DATA_BLOCK "DB_Result"
{ S7_Optimized_Access := 'TRUE' }
VERSION : 0.1
NON_RETAIN
   VAR
      TruePositive : Int;
      TrueNegative : Int;
      FalsePositive : Int;
      FalseNegative : Int;
      Predicted_class : Int;
      MismatchCount : Int;
      EXPECTED_TRUE_NEGATIVE : Int;
      EXPECTED_FALSE_POSITIVE : Int;
      EXPECTED_FALSE_NEGATIVE : Int;
      EXPECTED_TRUE_POSITIVE : Int;
      EXPECTED_PREDICITON_COUNT : Int;
      THRESHOLD : Real;
   END_VAR


BEGIN
   EXPECTED_TRUE_NEGATIVE := 1648;
   EXPECTED_FALSE_POSITIVE := 106;
   EXPECTED_FALSE_NEGATIVE := 55;
   EXPECTED_TRUE_POSITIVE := 885;
   EXPECTED_PREDICITON_COUNT := 2694;
   THRESHOLD := 0.05268643;

END_DATA_BLOCK

DATA_BLOCK "DB_Main"
{ S7_Optimized_Access := 'TRUE' }
VERSION : 0.1
NON_RETAIN
   VAR
      iState : Int;
      PredictCount : Int;
      bStart : Bool;
      Mse : Real;
   END_VAR


BEGIN

END_DATA_BLOCK

DATA_BLOCK "DB_Attack_v0_first_attack"
{ S7_Optimized_Access := 'TRUE' }
VERSION : 0.1
NON_RETAIN
   VAR
      DATA : Array[0..2693, 0..40] of Real;
   END_VAR


BEGIN
   DATA[0,0] := 2.427057;
   DATA[0,1] := 522.8467;
   DATA[0,2] := 2.0;
   DATA[0,3] := 2.0;
   DATA[0,4] := 262.0161;
   DATA[0,5] := 8.396437;
   DATA[0,6] := 328.6337;
   DATA[0,7] := 2.445391;
   DATA[0,8] := 2.0;
   DATA[0,9] := 2.0;
   DATA[0,10] := 2.0;
   DATA[0,11] := 19.74838;
   DATA[0,12] := 2.206835;
   DATA[0,13] := 956.1651;
   DATA[0,14] := 1.0;
   DATA[0,15] := 2.0;
   DATA[0,16] := 1.0;
   DATA[0,17] := 1.0;
   DATA[0,18] := 1.0;
   DATA[0,19] := 2.0;
   DATA[0,20] := 148.808;
   DATA[0,21] := 156.0882;
   DATA[0,22] := 1.713517;
   DATA[0,23] := 942.0662;
   DATA[0,24] := 2.0;
   DATA[0,25] := 2.0;
   DATA[0,26] := 7.878621;
   DATA[0,27] := 145.1166;
   DATA[0,28] := 264.5475;
   DATA[0,29] := 12.03538;
   DATA[0,30] := 1.723789;
   DATA[0,31] := 1.279621;
   DATA[0,32] := 0.7352687;
   DATA[0,33] := 0.3077859;
   DATA[0,34] := 2.0;
   DATA[0,35] := 250.8652;
   DATA[0,36] := 1.649953;
   DATA[0,37] := 189.5988;
   DATA[0,38] := 0.000128152;
   DATA[0,39] := 1.0;
   DATA[1,0] := 2.446274;
   DATA[1,1] := 522.886;
   DATA[1,2] := 2.0;
   DATA[1,3] := 2.0;
   DATA[1,4] := 262.0161;
   DATA[1,5] := 8.396437;
   DATA[1,6] := 328.6337;
   DATA[1,7] := 2.445391;
   DATA[1,8] := 2.0;
   DATA[1,9] := 2.0;
   DATA[1,10] := 2.0;
   DATA[1,11] := 19.74838;
   DATA[1,12] := 2.208244;
   DATA[1,13] := 956.1651;
   DATA[1,14] := 1.0;
   DATA[1,15] := 2.0;
   DATA[1,16] := 1.0;
   DATA[1,17] := 1.0;
   DATA[1,18] := 1.0;
   DATA[1,19] := 2.0;
   DATA[1,20] := 148.808;
   DATA[1,21] := 156.0882;
   DATA[1,22] := 1.715952;
   DATA[1,23] := 942.0277;
   DATA[1,24] := 2.0;
   DATA[1,25] := 2.0;
   DATA[1,26] := 7.878621;
   DATA[1,27] := 145.1166;
   DATA[1,28] := 264.5475;
   DATA[1,29] := 12.03538;
   DATA[1,30] := 1.723789;
   DATA[1,31] := 1.297554;
   DATA[1,32] := 0.7352687;
   DATA[1,33] := 0.3077859;
   DATA[1,34] := 2.0;
   DATA[1,35] := 250.8652;
   DATA[1,36] := 1.649953;
   DATA[1,37] := 189.6789;
   DATA[1,38] := 0.000128152;
   DATA[1,39] := 1.0;
   DATA[2,0] := 2.489191;
   DATA[2,1] := 522.8467;
   DATA[2,2] := 2.0;
   DATA[2,3] := 2.0;
   DATA[2,4] := 262.0161;
   DATA[2,5] := 8.394514;
   DATA[2,6] := 328.6337;
   DATA[2,7] := 2.442316;
   DATA[2,8] := 2.0;
   DATA[2,9] := 2.0;
   DATA[2,10] := 2.0;
   DATA[2,11] := 19.69076;
   DATA[2,12] := 2.208628;
   DATA[2,13] := 956.4855;
   DATA[2,14] := 1.0;
   DATA[2,15] := 2.0;
   DATA[2,16] := 1.0;
   DATA[2,17] := 1.0;
   DATA[2,18] := 1.0;
   DATA[2,19] := 2.0;
   DATA[2,20] := 148.808;
   DATA[2,21] := 156.0882;
   DATA[2,22] := 1.715952;
   DATA[2,23] := 941.8739;
   DATA[2,24] := 2.0;
   DATA[2,25] := 2.0;
   DATA[2,26] := 7.878621;
   DATA[2,27] := 145.1166;
   DATA[2,28] := 264.5475;
   DATA[2,29] := 12.03538;
   DATA[2,30] := 1.723404;
   DATA[2,31] := 1.293967;
   DATA[2,32] := 0.7352687;
   DATA[2,33] := 0.3086186;
   DATA[2,34] := 2.0;
   DATA[2,35] := 250.8812;
   DATA[2,36] := 1.649953;
   DATA[2,37] := 189.6789;
   DATA[2,38] := 0.000128152;
   DATA[2,39] := 1.0;
   DATA[3,0] := 2.53435;
   DATA[3,1] := 522.9645;
   DATA[3,2] := 2.0;
   DATA[3,3] := 2.0;
   DATA[3,4] := 262.0161;
   DATA[3,5] := 8.394514;
   DATA[3,6] := 328.6337;
   DATA[3,7] := 2.442316;
   DATA[3,8] := 2.0;
   DATA[3,9] := 2.0;
   DATA[3,10] := 2.0;
   DATA[3,11] := 19.69076;
   DATA[3,12] := 2.208628;
   DATA[3,13] := 956.806;
   DATA[3,14] := 1.0;
   DATA[3,15] := 2.0;
   DATA[3,16] := 1.0;
   DATA[3,17] := 1.0;
   DATA[3,18] := 1.0;
   DATA[3,19] := 2.0;
   DATA[3,20] := 148.808;
   DATA[3,21] := 156.0882;
   DATA[3,22] := 1.71467;
   DATA[3,23] := 941.797;
   DATA[3,24] := 2.0;
   DATA[3,25] := 2.0;
   DATA[3,26] := 7.878621;
   DATA[3,27] := 145.0141;
   DATA[3,28] := 264.5475;
   DATA[3,29] := 12.03538;
   DATA[3,30] := 1.723404;
   DATA[3,31] := 1.281158;
   DATA[3,32] := 0.7352687;
   DATA[3,33] := 0.3086186;
   DATA[3,34] := 2.0;
   DATA[3,35] := 250.8812;
   DATA[3,36] := 1.649953;
   DATA[3,37] := 189.6148;
   DATA[3,38] := 0.000128152;
   DATA[3,39] := 1.0;
   DATA[4,0] := 2.56926;
   DATA[4,1] := 523.4748;
   DATA[4,2] := 2.0;
   DATA[4,3] := 2.0;
   DATA[4,4] := 262.0161;
   DATA[4,5] := 8.394514;
   DATA[4,6] := 328.6337;
   DATA[4,7] := 2.443085;
   DATA[4,8] := 2.0;
   DATA[4,9] := 2.0;
   DATA[4,10] := 2.0;
   DATA[4,11] := 19.69076;
   DATA[4,12] := 2.208628;
   DATA[4,13] := 957.0864;
   DATA[4,14] := 1.0;
   DATA[4,15] := 2.0;
   DATA[4,16] := 1.0;
   DATA[4,17] := 1.0;
   DATA[4,18] := 1.0;
   DATA[4,19] := 2.0;
   DATA[4,20] := 148.808;
   DATA[4,21] := 156.0882;
   DATA[4,22] := 1.71467;
   DATA[4,23] := 942.22;
   DATA[4,24] := 2.0;
   DATA[4,25] := 2.0;
   DATA[4,26] := 7.878621;
   DATA[4,27] := 144.8859;
   DATA[4,28] := 264.5475;
   DATA[4,29] := 12.03538;
   DATA[4,30] := 1.723404;
   DATA[4,31] := 1.281158;
   DATA[4,32] := 0.7352687;
   DATA[4,33] := 0.3086186;
   DATA[4,34] := 2.0;
   DATA[4,35] := 250.8812;
   DATA[4,36] := 1.649953;
   DATA[4,37] := 189.5027;
   DATA[4,38] := 0.000128152;
   DATA[4,39] := 1.0;
   DATA[5,0] := 2.609294;
   DATA[5,1] := 523.8673;
   DATA[5,2] := 2.0;
   DATA[5,3] := 2.0;
   DATA[5,4] := 262.0161;
   DATA[5,5] := 8.394514;
   DATA[5,6] := 328.6337;
   DATA[5,7] := 2.44411;
   DATA[5,8] := 2.0;
   DATA[5,9] := 2.0;
   DATA[5,10] := 2.0;
   DATA[5,11] := 19.69076;
   DATA[5,12] := 2.207347;
   DATA[5,13] := 957.1664;
   DATA[5,14] := 1.0;
   DATA[5,15] := 2.0;
   DATA[5,16] := 1.0;
   DATA[5,17] := 1.0;
   DATA[5,18] := 1.0;
   DATA[5,19] := 2.0;
   DATA[5,20] := 148.808;
   DATA[5,21] := 155.96;
   DATA[5,22] := 1.71467;
   DATA[5,23] := 942.6429;
   DATA[5,24] := 2.0;
   DATA[5,25] := 2.0;
   DATA[5,26] := 7.878621;
   DATA[5,27] := 144.8859;
   DATA[5,28] := 264.5475;
   DATA[5,29] := 12.03538;
   DATA[5,30] := 1.723404;
   DATA[5,31] := 1.272704;
   DATA[5,32] := 0.7352687;
   DATA[5,33] := 0.3086186;
   DATA[5,34] := 2.0;
   DATA[5,35] := 250.753;
   DATA[5,36] := 1.649953;
   DATA[5,37] := 189.5027;
   DATA[5,38] := 0.000128152;
   DATA[5,39] := 1.0;
   DATA[6,0] := 2.637158;
   DATA[6,1] := 524.1028;
   DATA[6,2] := 2.0;
   DATA[6,3] := 2.0;
   DATA[6,4] := 262.0161;
   DATA[6,5] := 8.394514;
   DATA[6,6] := 328.6337;
   DATA[6,7] := 2.44411;
   DATA[6,8] := 2.0;
   DATA[6,9] := 2.0;
   DATA[6,10] := 2.0;
   DATA[6,11] := 19.69076;
   DATA[6,12] := 2.210037;
   DATA[6,13] := 957.0062;
   DATA[6,14] := 1.0;
   DATA[6,15] := 2.0;
   DATA[6,16] := 1.0;
   DATA[6,17] := 1.0;
   DATA[6,18] := 1.0;
   DATA[6,19] := 2.0;
   DATA[6,20] := 148.808;
   DATA[6,21] := 155.96;
   DATA[6,22] := 1.713004;
   DATA[6,23] := 942.7582;
   DATA[6,24] := 2.0;
   DATA[6,25] := 2.0;
   DATA[6,26] := 7.878621;
   DATA[6,27] := 144.8859;
   DATA[6,28] := 264.5475;
   DATA[6,29] := 12.03538;
   DATA[6,30] := 1.723404;
   DATA[6,31] := 1.270142;
   DATA[6,32] := 0.7352687;
   DATA[6,33] := 0.3086186;
   DATA[6,34] := 2.0;
   DATA[6,35] := 250.5928;
   DATA[6,36] := 1.649953;
   DATA[6,37] := 189.5027;
   DATA[6,38] := 0.000128152;
   DATA[6,39] := 1.0;
   DATA[7,0] := 2.652211;
   DATA[7,1] := 524.2206;
   DATA[7,2] := 2.0;
   DATA[7,3] := 2.0;
   DATA[7,4] := 262.0161;
   DATA[7,5] := 8.394514;
   DATA[7,6] := 328.6337;
   DATA[7,7] := 2.441803;
   DATA[7,8] := 2.0;
   DATA[7,9] := 2.0;
   DATA[7,10] := 2.0;
   DATA[7,11] := 19.69076;
   DATA[7,12] := 2.210037;
   DATA[7,13] := 957.2866;
   DATA[7,14] := 1.0;
   DATA[7,15] := 2.0;
   DATA[7,16] := 1.0;
   DATA[7,17] := 1.0;
   DATA[7,18] := 1.0;
   DATA[7,19] := 2.0;
   DATA[7,20] := 148.808;
   DATA[7,21] := 155.96;
   DATA[7,22] := 1.713004;
   DATA[7,23] := 943.1043;
   DATA[7,24] := 2.0;
   DATA[7,25] := 2.0;
   DATA[7,26] := 7.878621;
   DATA[7,27] := 144.8859;
   DATA[7,28] := 264.5475;
   DATA[7,29] := 12.03538;
   DATA[7,30] := 1.723404;
   DATA[7,31] := 1.262329;
   DATA[7,32] := 0.7352687;
   DATA[7,33] := 0.3086186;
   DATA[7,34] := 2.0;
   DATA[7,35] := 250.5928;
   DATA[7,36] := 1.649953;
   DATA[7,37] := 189.5027;
   DATA[7,38] := 0.000128152;
   DATA[7,39] := 1.0;
   DATA[8,0] := 2.655735;
   DATA[8,1] := 524.4954;
   DATA[8,2] := 2.0;
   DATA[8,3] := 2.0;
   DATA[8,4] := 262.0161;
   DATA[8,5] := 8.394514;
   DATA[8,6] := 328.6337;
   DATA[8,7] := 2.441803;
   DATA[8,8] := 2.0;
   DATA[8,9] := 2.0;
   DATA[8,10] := 2.0;
   DATA[8,11] := 19.66195;
   DATA[8,12] := 2.210037;
   DATA[8,13] := 957.6071;
   DATA[8,14] := 1.0;
   DATA[8,15] := 2.0;
   DATA[8,16] := 1.0;
   DATA[8,17] := 1.0;
   DATA[8,18] := 1.0;
   DATA[8,19] := 2.0;
   DATA[8,20] := 148.808;
   DATA[8,21] := 155.96;
   DATA[8,22] := 1.71262;
   DATA[8,23] := 943.3735;
   DATA[8,24] := 2.0;
   DATA[8,25] := 2.0;
   DATA[8,26] := 7.878621;
   DATA[8,27] := 144.8859;
   DATA[8,28] := 264.5475;
   DATA[8,29] := 12.03538;
   DATA[8,30] := 1.723404;
   DATA[8,31] := 1.270398;
   DATA[8,32] := 0.7352687;
   DATA[8,33] := 0.3086186;
   DATA[8,34] := 2.0;
   DATA[8,35] := 250.9132;
   DATA[8,36] := 1.649953;
   DATA[8,37] := 189.5027;
   DATA[8,38] := 0.000128152;
   DATA[8,39] := 1.0;
   DATA[9,0] := 2.64997;
   DATA[9,1] := 524.0636;
   DATA[9,2] := 2.0;
   DATA[9,3] := 2.0;
   DATA[9,4] := 262.0161;
   DATA[9,5] := 8.394514;
   DATA[9,6] := 328.6337;
   DATA[9,7] := 2.441803;
   DATA[9,8] := 2.0;
   DATA[9,9] := 2.0;
   DATA[9,10] := 2.0;
   DATA[9,11] := 19.66195;
   DATA[9,12] := 2.210037;
   DATA[9,13] := 957.2866;
   DATA[9,14] := 1.0;
   DATA[9,15] := 2.0;
   DATA[9,16] := 1.0;
   DATA[9,17] := 1.0;
   DATA[9,18] := 1.0;
   DATA[9,19] := 2.0;
   DATA[9,20] := 148.808;
   DATA[9,21] := 155.96;
   DATA[9,22] := 1.71262;
   DATA[9,23] := 943.6042;
   DATA[9,24] := 2.0;
   DATA[9,25] := 2.0;
   DATA[9,26] := 7.878621;
   DATA[9,27] := 144.8859;
   DATA[9,28] := 264.5475;
   DATA[9,29] := 12.03538;
   DATA[9,30] := 1.726224;
   DATA[9,31] := 1.281158;
   DATA[9,32] := 0.7352687;
   DATA[9,33] := 0.3084905;
   DATA[9,34] := 2.0;
   DATA[9,35] := 250.9132;
   DATA[9,36] := 1.649953;
   DATA[9,37] := 189.5668;
   DATA[9,38] := 0.000128152;
   DATA[9,39] := 1.0;
   DATA[10,0] := 2.630433;
   DATA[10,1] := 524.1028;
   DATA[10,2] := 2.0;
   DATA[10,3] := 2.0;
   DATA[10,4] := 262.0161;
   DATA[10,5] := 8.394514;
   DATA[10,6] := 328.6337;
   DATA[10,7] := 2.441803;
   DATA[10,8] := 2.0;
   DATA[10,9] := 2.0;
   DATA[10,10] := 2.0;
   DATA[10,11] := 19.68756;
   DATA[10,12] := 2.210037;
   DATA[10,13] := 957.6071;
   DATA[10,14] := 1.0;
   DATA[10,15] := 2.0;
   DATA[10,16] := 1.0;
   DATA[10,17] := 1.0;
   DATA[10,18] := 1.0;
   DATA[10,19] := 2.0;
   DATA[10,20] := 148.808;
   DATA[10,21] := 155.96;
   DATA[10,22] := 1.715439;
   DATA[10,23] := 943.9118;
   DATA[10,24] := 2.0;
   DATA[10,25] := 2.0;
   DATA[10,26] := 7.878621;
   DATA[10,27] := 144.8859;
   DATA[10,28] := 264.5475;
   DATA[10,29] := 12.03538;
   DATA[10,30] := 1.726352;
   DATA[10,31] := 1.276162;
   DATA[10,32] := 0.7352687;
   DATA[10,33] := 0.3081062;
   DATA[10,34] := 2.0;
   DATA[10,35] := 251.1055;
   DATA[10,36] := 1.649953;
   DATA[10,37] := 189.8231;
   DATA[10,38] := 0.000128152;
   DATA[10,39] := 1.0;
   DATA[11,0] := 2.621785;
   DATA[11,1] := 523.7496;
   DATA[11,2] := 2.0;
   DATA[11,3] := 2.0;
   DATA[11,4] := 262.0161;
   DATA[11,5] := 8.391951;
   DATA[11,6] := 328.6337;
   DATA[11,7] := 2.441803;
   DATA[11,8] := 2.0;
   DATA[11,9] := 2.0;
   DATA[11,10] := 2.0;
   DATA[11,11] := 19.72598;
   DATA[11,12] := 2.210037;
   DATA[11,13] := 957.2065;
   DATA[11,14] := 1.0;
   DATA[11,15] := 2.0;
   DATA[11,16] := 1.0;
   DATA[11,17] := 1.0;
   DATA[11,18] := 1.0;
   DATA[11,19] := 2.0;
   DATA[11,20] := 148.808;
   DATA[11,21] := 156.1138;
   DATA[11,22] := 1.716721;
   DATA[11,23] := 943.9118;
   DATA[11,24] := 2.0;
   DATA[11,25] := 2.0;
   DATA[11,26] := 7.878621;
   DATA[11,27] := 144.8859;
   DATA[11,28] := 264.5475;
   DATA[11,29] := 12.03538;
   DATA[11,30] := 1.726352;
   DATA[11,31] := 1.282183;
   DATA[11,32] := 0.7352687;
   DATA[11,33] := 0.3074016;
   DATA[11,34] := 2.0;
   DATA[11,35] := 251.1856;
   DATA[11,36] := 1.649953;
   DATA[11,37] := 189.9994;
   DATA[11,38] := 0.000128152;
   DATA[11,39] := 1.0;
   DATA[12,0] := 2.61602;
   DATA[12,1] := 523.4355;
   DATA[12,2] := 2.0;
   DATA[12,3] := 2.0;
   DATA[12,4] := 262.0161;
   DATA[12,5] := 8.390669;
   DATA[12,6] := 328.6337;
   DATA[12,7] := 2.441803;
   DATA[12,8] := 2.0;
   DATA[12,9] := 2.0;
   DATA[12,10] := 2.0;
   DATA[12,11] := 19.75479;
   DATA[12,12] := 2.210037;
   DATA[12,13] := 957.5269;
   DATA[12,14] := 1.0;
   DATA[12,15] := 2.0;
   DATA[12,16] := 1.0;
   DATA[12,17] := 1.0;
   DATA[12,18] := 1.0;
   DATA[12,19] := 2.0;
   DATA[12,20] := 148.808;
   DATA[12,21] := 156.1138;
   DATA[12,22] := 1.717874;
   DATA[12,23] := 944.181;
   DATA[12,24] := 2.0;
   DATA[12,25] := 2.0;
   DATA[12,26] := 7.878621;
   DATA[12,27] := 144.8859;
   DATA[12,28] := 264.5475;
   DATA[12,29] := 12.03538;
   DATA[12,30] := 1.72725;
   DATA[12,31] := 1.275778;
   DATA[12,32] := 0.7352687;
   DATA[12,33] := 0.3066329;
   DATA[12,34] := 2.0;
   DATA[12,35] := 251.1856;
   DATA[12,36] := 1.649953;
   DATA[12,37] := 189.9994;
   DATA[12,38] := 0.000128152;
   DATA[12,39] := 1.0;
   DATA[13,0] := 2.599366;
   DATA[13,1] := 523.043;
   DATA[13,2] := 2.0;
   DATA[13,3] := 2.0;
   DATA[13,4] := 262.0161;
   DATA[13,5] := 8.390669;
   DATA[13,6] := 328.6337;
   DATA[13,7] := 2.441803;
   DATA[13,8] := 2.0;
   DATA[13,9] := 2.0;
   DATA[13,10] := 2.0;
   DATA[13,11] := 19.79;
   DATA[13,12] := 2.210037;
   DATA[13,13] := 957.8875;
   DATA[13,14] := 1.0;
   DATA[13,15] := 2.0;
   DATA[13,16] := 1.0;
   DATA[13,17] := 1.0;
   DATA[13,18] := 1.0;
   DATA[13,19] := 2.0;
   DATA[13,20] := 148.808;
   DATA[13,21] := 156.1138;
   DATA[13,22] := 1.717874;
   DATA[13,23] := 943.9118;
   DATA[13,24] := 2.0;
   DATA[13,25] := 2.0;
   DATA[13,26] := 7.878621;
   DATA[13,27] := 144.8859;
   DATA[13,28] := 264.5475;
   DATA[13,29] := 12.03538;
   DATA[13,30] := 1.728275;
   DATA[13,31] := 1.272192;
   DATA[13,32] := 0.7352687;
   DATA[13,33] := 0.3066329;
   DATA[13,34] := 2.0;
   DATA[13,35] := 251.1856;
   DATA[13,36] := 1.649953;
   DATA[13,37] := 189.9994;
   DATA[13,38] := 0.000128152;
   DATA[13,39] := 1.0;
   DATA[14,0] := 2.588476;
   DATA[14,1] := 522.729;
   DATA[14,2] := 2.0;
   DATA[14,3] := 2.0;
   DATA[14,4] := 262.0161;
   DATA[14,5] := 8.390669;
   DATA[14,6] := 328.6337;
   DATA[14,7] := 2.441803;
   DATA[14,8] := 2.0;
   DATA[14,9] := 2.0;
   DATA[14,10] := 2.0;
   DATA[14,11] := 19.79;
   DATA[14,12] := 2.209525;
   DATA[14,13] := 958.288;
   DATA[14,14] := 1.0;
   DATA[14,15] := 2.0;
   DATA[14,16] := 1.0;
   DATA[14,17] := 1.0;
   DATA[14,18] := 1.0;
   DATA[14,19] := 2.0;
   DATA[14,20] := 148.808;
   DATA[14,21] := 156.1138;
   DATA[14,22] := 1.717874;
   DATA[14,23] := 943.9887;
   DATA[14,24] := 2.0;
   DATA[14,25] := 2.0;
   DATA[14,26] := 7.878621;
   DATA[14,27] := 144.8859;
   DATA[14,28] := 264.5475;
   DATA[14,29] := 12.26609;
   DATA[14,30] := 1.728275;
   DATA[14,31] := 1.282951;
   DATA[14,32] := 0.7352687;
   DATA[14,33] := 0.3066329;
   DATA[14,34] := 2.0;
   DATA[14,35] := 251.1856;
   DATA[14,36] := 1.649953;
   DATA[14,37] := 189.9994;
   DATA[14,38] := 0.000128152;
   DATA[14,39] := 1.0;
   DATA[15,0] := 2.567979;
   DATA[15,1] := 522.6505;
   DATA[15,2] := 2.0;
   DATA[15,3] := 2.0;
   DATA[15,4] := 262.0161;
   DATA[15,5] := 8.390669;
   DATA[15,6] := 328.6337;
   DATA[15,7] := 2.441803;
   DATA[15,8] := 2.0;
   DATA[15,9] := 2.0;
   DATA[15,10] := 2.0;
   DATA[15,11] := 19.73878;
   DATA[15,12] := 2.209525;
   DATA[15,13] := 958.288;
   DATA[15,14] := 1.0;
   DATA[15,15] := 2.0;
   DATA[15,16] := 1.0;
   DATA[15,17] := 1.0;
   DATA[15,18] := 1.0;
   DATA[15,19] := 2.0;
   DATA[15,20] := 148.808;
   DATA[15,21] := 156.1138;
   DATA[15,22] := 1.717874;
   DATA[15,23] := 944.4117;
   DATA[15,24] := 2.0;
   DATA[15,25] := 2.0;
   DATA[15,26] := 7.878621;
   DATA[15,27] := 144.8859;
   DATA[15,28] := 264.5475;
   DATA[15,29] := 12.26609;
   DATA[15,30] := 1.728275;
   DATA[15,31] := 1.282951;
   DATA[15,32] := 0.7352687;
   DATA[15,33] := 0.3066329;
   DATA[15,34] := 2.0;
   DATA[15,35] := 251.1856;
   DATA[15,36] := 1.649953;
   DATA[15,37] := 189.9994;
   DATA[15,38] := 0.000128152;
   DATA[15,39] := 1.0;
   DATA[16,0] := 2.556769;
   DATA[16,1] := 522.6897;
   DATA[16,2] := 2.0;
   DATA[16,3] := 2.0;
   DATA[16,4] := 262.0161;
   DATA[16,5] := 8.390669;
   DATA[16,6] := 328.6337;
   DATA[16,7] := 2.441803;
   DATA[16,8] := 2.0;
   DATA[16,9] := 2.0;
   DATA[16,10] := 2.0;
   DATA[16,11] := 19.70997;
   DATA[16,12] := 2.207091;
   DATA[16,13] := 958.5684;
   DATA[16,14] := 1.0;
   DATA[16,15] := 2.0;
   DATA[16,16] := 1.0;
   DATA[16,17] := 1.0;
   DATA[16,18] := 1.0;
   DATA[16,19] := 2.0;
   DATA[16,20] := 148.808;
   DATA[16,21] := 156.1138;
   DATA[16,22] := 1.717874;
   DATA[16,23] := 944.527;
   DATA[16,24] := 2.0;
   DATA[16,25] := 2.0;
   DATA[16,26] := 7.878621;
   DATA[16,27] := 144.8859;
   DATA[16,28] := 264.5475;
   DATA[16,29] := 12.26609;
   DATA[16,30] := 1.729172;
   DATA[16,31] := 1.291533;
   DATA[16,32] := 0.7373172;
   DATA[16,33] := 0.3066329;
   DATA[16,34] := 2.0;
   DATA[16,35] := 251.1856;
   DATA[16,36] := 1.649953;
   DATA[16,37] := 189.8872;
   DATA[16,38] := 0.000128152;
   DATA[16,39] := 1.0;
   DATA[17,0] := 2.53435;
   DATA[17,1] := 522.6897;
   DATA[17,2] := 2.0;
   DATA[17,3] := 2.0;
   DATA[17,4] := 262.0161;
   DATA[17,5] := 8.390669;
   DATA[17,6] := 328.6081;
   DATA[17,7] := 2.439881;
   DATA[17,8] := 2.0;
   DATA[17,9] := 2.0;
   DATA[17,10] := 2.0;
   DATA[17,11] := 19.68756;
   DATA[17,12] := 2.20581;
   DATA[17,13] := 958.7286;
   DATA[17,14] := 1.0;
   DATA[17,15] := 2.0;
   DATA[17,16] := 1.0;
   DATA[17,17] := 1.0;
   DATA[17,18] := 1.0;
   DATA[17,19] := 2.0;
   DATA[17,20] := 148.808;
   DATA[17,21] := 156.1138;
   DATA[17,22] := 1.716464;
   DATA[17,23] := 944.7962;
   DATA[17,24] := 2.0;
   DATA[17,25] := 2.0;
   DATA[17,26] := 7.878621;
   DATA[17,27] := 144.8859;
   DATA[17,28] := 264.5475;
   DATA[17,29] := 12.26609;
   DATA[17,30] := 1.729172;
   DATA[17,31] := 1.291533;
   DATA[17,32] := 0.7385975;
   DATA[17,33] := 0.30785;
   DATA[17,34] := 2.0;
   DATA[17,35] := 251.1856;
   DATA[17,36] := 1.649953;
   DATA[17,37] := 189.8872;
   DATA[17,38] := 0.000128152;
   DATA[17,39] := 1.0;
   DATA[18,0] := 2.521859;
   DATA[18,1] := 522.6505;
   DATA[18,2] := 2.0;
   DATA[18,3] := 2.0;
   DATA[18,4] := 262.0161;
   DATA[18,5] := 8.390669;
   DATA[18,6] := 328.3773;
   DATA[18,7] := 2.439881;
   DATA[18,8] := 2.0;
   DATA[18,9] := 2.0;
   DATA[18,10] := 2.0;
   DATA[18,11] := 19.68756;
   DATA[18,12] := 2.205426;
   DATA[18,13] := 958.4882;
   DATA[18,14] := 1.0;
   DATA[18,15] := 2.0;
   DATA[18,16] := 1.0;
   DATA[18,17] := 1.0;
   DATA[18,18] := 1.0;
   DATA[18,19] := 2.0;
   DATA[18,20] := 148.808;
   DATA[18,21] := 156.1138;
   DATA[18,22] := 1.71608;
   DATA[18,23] := 945.4499;
   DATA[18,24] := 2.0;
   DATA[18,25] := 2.0;
   DATA[18,26] := 7.878621;
   DATA[18,27] := 144.8859;
   DATA[18,28] := 264.5475;
   DATA[18,29] := 12.26609;
   DATA[18,30] := 1.729172;
   DATA[18,31] := 1.284745;
   DATA[18,32] := 0.7385975;
   DATA[18,33] := 0.3083624;
   DATA[18,34] := 2.0;
   DATA[18,35] := 251.1856;
   DATA[18,36] := 1.649953;
   DATA[18,37] := 189.8872;
   DATA[18,38] := 0.000128152;
   DATA[18,39] := 1.0;
   DATA[19,0] := 2.502642;
   DATA[19,1] := 522.6897;
   DATA[19,2] := 2.0;
   DATA[19,3] := 2.0;
   DATA[19,4] := 262.0161;
   DATA[19,5] := 8.390669;
   DATA[19,6] := 328.3773;
   DATA[19,7] := 2.439881;
   DATA[19,8] := 2.0;
   DATA[19,9] := 2.0;
   DATA[19,10] := 2.0;
   DATA[19,11] := 19.68756;
   DATA[19,12] := 2.205426;
   DATA[19,13] := 958.5684;
   DATA[19,14] := 1.0;
   DATA[19,15] := 2.0;
   DATA[19,16] := 1.0;
   DATA[19,17] := 1.0;
   DATA[19,18] := 1.0;
   DATA[19,19] := 2.0;
   DATA[19,20] := 148.808;
   DATA[19,21] := 156.1138;
   DATA[19,22] := 1.715824;
   DATA[19,23] := 945.5268;
   DATA[19,24] := 2.0;
   DATA[19,25] := 2.0;
   DATA[19,26] := 7.878621;
   DATA[19,27] := 144.8859;
   DATA[19,28] := 264.5475;
   DATA[19,29] := 12.26609;
   DATA[19,30] := 1.729172;
   DATA[19,31] := 1.288203;
   DATA[19,32] := 0.7385975;
   DATA[19,33] := 0.3083624;
   DATA[19,34] := 2.0;
   DATA[19,35] := 251.1856;
   DATA[19,36] := 1.649953;
   DATA[19,37] := 189.8872;
   DATA[19,38] := 0.000128152;
   DATA[19,39] := 1.0;
   DATA[20,0] := 2.489191;
   DATA[20,1] := 522.729;
   DATA[20,2] := 2.0;
   DATA[20,3] := 2.0;
   DATA[20,4] := 262.0161;
   DATA[20,5] := 8.390669;
   DATA[20,6] := 328.3773;
   DATA[20,7] := 2.439881;
   DATA[20,8] := 2.0;
   DATA[20,9] := 2.0;
   DATA[20,10] := 2.0;
   DATA[20,11] := 19.68756;
   DATA[20,12] := 2.207347;
   DATA[20,13] := 958.8087;
   DATA[20,14] := 1.0;
   DATA[20,15] := 2.0;
   DATA[20,16] := 1.0;
   DATA[20,17] := 1.0;
   DATA[20,18] := 1.0;
   DATA[20,19] := 2.0;
   DATA[20,20] := 148.808;
   DATA[20,21] := 156.1138;
   DATA[20,22] := 1.715824;
   DATA[20,23] := 945.6806;
   DATA[20,24] := 2.0;
   DATA[20,25] := 2.0;
   DATA[20,26] := 7.878621;
   DATA[20,27] := 144.8859;
   DATA[20,28] := 264.5475;
   DATA[20,29] := 12.11228;
   DATA[20,30] := 1.729172;
   DATA[20,31] := 1.282823;
   DATA[20,32] := 0.7385975;
   DATA[20,33] := 0.3083624;
   DATA[20,34] := 2.0;
   DATA[20,35] := 251.1856;
   DATA[20,36] := 1.649953;
   DATA[20,37] := 189.8872;
   DATA[20,38] := 0.000128152;
   DATA[20,39] := 1.0;
   DATA[21,0] := 2.473497;
   DATA[21,1] := 522.5327;
   DATA[21,2] := 2.0;
   DATA[21,3] := 2.0;
   DATA[21,4] := 262.0161;
   DATA[21,5] := 8.390669;
   DATA[21,6] := 328.6337;
   DATA[21,7] := 2.439881;
   DATA[21,8] := 2.0;
   DATA[21,9] := 2.0;
   DATA[21,10] := 2.0;
   DATA[21,11] := 19.68756;
   DATA[21,12] := 2.208628;
   DATA[21,13] := 958.5684;
   DATA[21,14] := 1.0;
   DATA[21,15] := 2.0;
   DATA[21,16] := 1.0;
   DATA[21,17] := 1.0;
   DATA[21,18] := 1.0;
   DATA[21,19] := 2.0;
   DATA[21,20] := 148.808;
   DATA[21,21] := 156.1138;
   DATA[21,22] := 1.715824;
   DATA[21,23] := 945.6806;
   DATA[21,24] := 2.0;
   DATA[21,25] := 2.0;
   DATA[21,26] := 7.878621;
   DATA[21,27] := 144.8859;
   DATA[21,28] := 264.5475;
   DATA[21,29] := 12.11228;
   DATA[21,30] := 1.729172;
   DATA[21,31] := 1.281286;
   DATA[21,32] := 0.7385975;
   DATA[21,33] := 0.3083624;
   DATA[21,34] := 2.0;
   DATA[21,35] := 251.1856;
   DATA[21,36] := 1.649953;
   DATA[21,37] := 189.8872;
   DATA[21,38] := 0.000128152;
   DATA[21,39] := 1.0;
   DATA[22,0] := 2.458764;
   DATA[22,1] := 522.886;
   DATA[22,2] := 2.0;
   DATA[22,3] := 2.0;
   DATA[22,4] := 262.0161;
   DATA[22,5] := 8.390669;
   DATA[22,6] := 328.6337;
   DATA[22,7] := 2.439881;
   DATA[22,8] := 2.0;
   DATA[22,9] := 2.0;
   DATA[22,10] := 2.0;
   DATA[22,11] := 19.57872;
   DATA[22,12] := 2.208628;
   DATA[22,13] := 958.6084;
   DATA[22,14] := 1.0;
   DATA[22,15] := 2.0;
   DATA[22,16] := 1.0;
   DATA[22,17] := 1.0;
   DATA[22,18] := 1.0;
   DATA[22,19] := 2.0;
   DATA[22,20] := 148.808;
   DATA[22,21] := 156.1138;
   DATA[22,22] := 1.717361;
   DATA[22,23] := 945.9498;
   DATA[22,24] := 2.0;
   DATA[22,25] := 2.0;
   DATA[22,26] := 7.878621;
   DATA[22,27] := 144.8859;
   DATA[22,28] := 264.5475;
   DATA[22,29] := 12.11228;
   DATA[22,30] := 1.729172;
   DATA[22,31] := 1.287306;
   DATA[22,32] := 0.7385975;
   DATA[22,33] := 0.3079781;
   DATA[22,34] := 2.0;
   DATA[22,35] := 251.1856;
   DATA[22,36] := 1.649953;
   DATA[22,37] := 189.8872;
   DATA[22,38] := 0.000128152;
   DATA[22,39] := 1.0;
   DATA[23,0] := 2.444031;
   DATA[23,1] := 523.4355;
   DATA[23,2] := 2.0;
   DATA[23,3] := 2.0;
   DATA[23,4] := 262.0161;
   DATA[23,5] := 8.390669;
   DATA[23,6] := 328.6337;
   DATA[23,7] := 2.439881;
   DATA[23,8] := 2.0;
   DATA[23,9] := 2.0;
   DATA[23,10] := 2.0;
   DATA[23,11] := 19.57232;
   DATA[23,12] := 2.208628;
   DATA[23,13] := 958.328;
   DATA[23,14] := 1.0;
   DATA[23,15] := 2.0;
   DATA[23,16] := 1.0;
   DATA[23,17] := 1.0;
   DATA[23,18] := 1.0;
   DATA[23,19] := 2.0;
   DATA[23,20] := 148.808;
   DATA[23,21] := 156.1138;
   DATA[23,22] := 1.718515;
   DATA[23,23] := 945.9498;
   DATA[23,24] := 2.0;
   DATA[23,25] := 2.0;
   DATA[23,26] := 7.878621;
   DATA[23,27] := 144.8859;
   DATA[23,28] := 264.5475;
   DATA[23,29] := 12.11228;
   DATA[23,30] := 1.729172;
   DATA[23,31] := 1.283464;
   DATA[23,32] := 0.7385975;
   DATA[23,33] := 0.3065689;
   DATA[23,34] := 2.0;
   DATA[23,35] := 251.1856;
   DATA[23,36] := 1.649953;
   DATA[23,37] := 189.8872;
   DATA[23,38] := 0.000128152;
   DATA[23,39] := 1.0;
   DATA[24,0] := 2.434744;
   DATA[24,1] := 523.671;
   DATA[24,2] := 2.0;
   DATA[24,3] := 2.0;
   DATA[24,4] := 262.0161;
   DATA[24,5] := 8.390669;
   DATA[24,6] := 328.6337;
   DATA[24,7] := 2.439881;
   DATA[24,8] := 2.0;
   DATA[24,9] := 2.0;
   DATA[24,10] := 2.0;
   DATA[24,11] := 19.55311;
   DATA[24,12] := 2.211318;
   DATA[24,13] := 958.368;
   DATA[24,14] := 1.0;
   DATA[24,15] := 2.0;
   DATA[24,16] := 1.0;
   DATA[24,17] := 1.0;
   DATA[24,18] := 1.0;
   DATA[24,19] := 2.0;
   DATA[24,20] := 148.808;
   DATA[24,21] := 156.1138;
   DATA[24,22] := 1.718515;
   DATA[24,23] := 946.1036;
   DATA[24,24] := 2.0;
   DATA[24,25] := 2.0;
   DATA[24,26] := 7.878621;
   DATA[24,27] := 144.8859;
   DATA[24,28] := 264.5475;
   DATA[24,29] := 12.11228;
   DATA[24,30] := 1.729172;
   DATA[24,31] := 1.282439;
   DATA[24,32] := 0.7385975;
   DATA[24,33] := 0.3065689;
   DATA[24,34] := 2.0;
   DATA[24,35] := 251.1856;
   DATA[24,36] := 1.649953;
   DATA[24,37] := 189.8872;
   DATA[24,38] := 0.000128152;
   DATA[24,39] := 1.0;
   DATA[25,0] := 2.423854;
   DATA[25,1] := 523.7496;
   DATA[25,2] := 2.0;
   DATA[25,3] := 2.0;
   DATA[25,4] := 262.0161;
   DATA[25,5] := 8.390669;
   DATA[25,6] := 328.6337;
   DATA[25,7] := 2.439881;
   DATA[25,8] := 2.0;
   DATA[25,9] := 2.0;
   DATA[25,10] := 2.0;
   DATA[25,11] := 19.55311;
   DATA[25,12] := 2.211318;
   DATA[25,13] := 958.1678;
   DATA[25,14] := 1.0;
   DATA[25,15] := 2.0;
   DATA[25,16] := 1.0;
   DATA[25,17] := 1.0;
   DATA[25,18] := 1.0;
   DATA[25,19] := 2.0;
   DATA[25,20] := 148.808;
   DATA[25,21] := 156.1138;
   DATA[25,22] := 1.718515;
   DATA[25,23] := 946.0267;
   DATA[25,24] := 2.0;
   DATA[25,25] := 2.0;
   DATA[25,26] := 7.878621;
   DATA[25,27] := 144.9116;
   DATA[25,28] := 264.5475;
   DATA[25,29] := 12.11228;
   DATA[25,30] := 1.729172;
   DATA[25,31] := 1.276547;
   DATA[25,32] := 0.7383414;
   DATA[25,33] := 0.3065689;
   DATA[25,34] := 2.0;
   DATA[25,35] := 251.1856;
   DATA[25,36] := 1.649953;
   DATA[25,37] := 189.8872;
   DATA[25,38] := 0.000128152;
   DATA[25,39] := 1.0;
   DATA[26,0] := 2.421932;
   DATA[26,1] := 523.8281;
   DATA[26,2] := 2.0;
   DATA[26,3] := 2.0;
   DATA[26,4] := 262.0161;
   DATA[26,5] := 8.390669;
   DATA[26,6] := 328.6337;
   DATA[26,7] := 2.439881;
   DATA[26,8] := 2.0;
   DATA[26,9] := 2.0;
   DATA[26,10] := 2.0;
   DATA[26,11] := 19.60433;
   DATA[26,12] := 2.211318;
   DATA[26,13] := 958.1277;
   DATA[26,14] := 1.0;
   DATA[26,15] := 2.0;
   DATA[26,16] := 1.0;
   DATA[26,17] := 1.0;
   DATA[26,18] := 1.0;
   DATA[26,19] := 2.0;
   DATA[26,20] := 148.808;
   DATA[26,21] := 156.1138;
   DATA[26,22] := 1.718515;
   DATA[26,23] := 946.2958;
   DATA[26,24] := 2.0;
   DATA[26,25] := 2.0;
   DATA[26,26] := 7.878621;
   DATA[26,27] := 144.9116;
   DATA[26,28] := 264.5475;
   DATA[26,29] := 12.11228;
   DATA[26,30] := 1.729172;
   DATA[26,31] := 1.265659;
   DATA[26,32] := 0.7379573;
   DATA[26,33] := 0.3065689;
   DATA[26,34] := 2.0;
   DATA[26,35] := 251.1856;
   DATA[26,36] := 1.649953;
   DATA[26,37] := 189.8872;
   DATA[26,38] := 0.000128152;
   DATA[26,39] := 1.0;
   DATA[27,0] := 2.425776;
   DATA[27,1] := 524.2598;
   DATA[27,2] := 2.0;
   DATA[27,3] := 2.0;
   DATA[27,4] := 262.0161;
   DATA[27,5] := 8.390669;
   DATA[27,6] := 328.6337;
   DATA[27,7] := 2.439881;
   DATA[27,8] := 2.0;
   DATA[27,9] := 2.0;
   DATA[27,10] := 2.0;
   DATA[27,11] := 19.60753;
   DATA[27,12] := 2.212215;
   DATA[27,13] := 958.0076;
   DATA[27,14] := 1.0;
   DATA[27,15] := 2.0;
   DATA[27,16] := 1.0;
   DATA[27,17] := 1.0;
   DATA[27,18] := 1.0;
   DATA[27,19] := 2.0;
   DATA[27,20] := 148.808;
   DATA[27,21] := 156.1138;
   DATA[27,22] := 1.718515;
   DATA[27,23] := 946.2958;
   DATA[27,24] := 2.0;
   DATA[27,25] := 2.0;
   DATA[27,26] := 7.878621;
   DATA[27,27] := 144.9116;
   DATA[27,28] := 264.5475;
   DATA[27,29] := 12.11228;
   DATA[27,30] := 1.728788;
   DATA[27,31] := 1.262457;
   DATA[27,32] := 0.7361649;
   DATA[27,33] := 0.3065689;
   DATA[27,34] := 2.0;
   DATA[27,35] := 251.1535;
   DATA[27,36] := 1.649953;
   DATA[27,37] := 189.8872;
   DATA[27,38] := 0.000128152;
   DATA[27,39] := 1.0;
   DATA[28,0] := 2.471575;
   DATA[28,1] := 524.1421;
   DATA[28,2] := 2.0;
   DATA[28,3] := 2.0;
   DATA[28,4] := 262.0161;
   DATA[28,5] := 8.390669;
   DATA[28,6] := 328.6337;
   DATA[28,7] := 2.439881;
   DATA[28,8] := 2.0;
   DATA[28,9] := 2.0;
   DATA[28,10] := 2.0;
   DATA[28,11] := 19.65555;
   DATA[28,12] := 2.212215;
   DATA[28,13] := 957.9275;
   DATA[28,14] := 1.0;
   DATA[28,15] := 2.0;
   DATA[28,16] := 1.0;
   DATA[28,17] := 1.0;
   DATA[28,18] := 1.0;
   DATA[28,19] := 2.0;
   DATA[28,20] := 148.808;
   DATA[28,21] := 156.1138;
   DATA[28,22] := 1.717361;
   DATA[28,23] := 946.2958;
   DATA[28,24] := 2.0;
   DATA[28,25] := 2.0;
   DATA[28,26] := 7.878621;
   DATA[28,27] := 144.9116;
   DATA[28,28] := 264.5475;
   DATA[28,29] := 12.11228;
   DATA[28,30] := 1.72725;
   DATA[28,31] := 1.27027;
   DATA[28,32] := 0.7357808;
   DATA[28,33] := 0.3065689;
   DATA[28,34] := 2.0;
   DATA[28,35] := 251.0414;
   DATA[28,36] := 1.649953;
   DATA[28,37] := 189.8872;
   DATA[28,38] := 0.000128152;
   DATA[28,39] := 1.0;
   DATA[29,0] := 2.527624;
   DATA[29,1] := 524.2598;
   DATA[29,2] := 2.0;
   DATA[29,3] := 2.0;
   DATA[29,4] := 262.0161;
   DATA[29,5] := 8.390669;
   DATA[29,6] := 328.6337;
   DATA[29,7] := 2.439881;
   DATA[29,8] := 2.0;
   DATA[29,9] := 2.0;
   DATA[29,10] := 2.0;
   DATA[29,11] := 19.68756;
   DATA[29,12] := 2.212215;
   DATA[29,13] := 957.6071;
   DATA[29,14] := 1.0;
   DATA[29,15] := 2.0;
   DATA[29,16] := 1.0;
   DATA[29,17] := 1.0;
   DATA[29,18] := 1.0;
   DATA[29,19] := 2.0;
   DATA[29,20] := 148.808;
   DATA[29,21] := 156.1138;
   DATA[29,22] := 1.717361;
   DATA[29,23] := 946.2958;
   DATA[29,24] := 2.0;
   DATA[29,25] := 2.0;
   DATA[29,26] := 7.878621;
   DATA[29,27] := 144.9116;
   DATA[29,28] := 264.5475;
   DATA[29,29] := 12.11228;
   DATA[29,30] := 1.72725;
   DATA[29,31] := 1.271551;
   DATA[29,32] := 0.7348846;
   DATA[29,33] := 0.3065689;
   DATA[29,34] := 2.0;
   DATA[29,35] := 251.0414;
   DATA[29,36] := 1.649953;
   DATA[29,37] := 189.8872;
   DATA[29,38] := 0.000128152;
   DATA[29,39] := 1.0;
   DATA[30,0] := 2.554847;
   DATA[30,1] := 524.6523;
   DATA[30,2] := 2.0;
   DATA[30,3] := 2.0;
   DATA[30,4] := 262.0161;
   DATA[30,5] := 8.390669;
   DATA[30,6] := 328.6337;
   DATA[30,7] := 2.439881;
   DATA[30,8] := 2.0;
   DATA[30,9] := 2.0;
   DATA[30,10] := 2.0;
   DATA[30,11] := 19.68756;
   DATA[30,12] := 2.212215;
   DATA[30,13] := 957.6871;
   DATA[30,14] := 1.0;
   DATA[30,15] := 2.0;
   DATA[30,16] := 1.0;
   DATA[30,17] := 1.0;
   DATA[30,18] := 1.0;
   DATA[30,19] := 2.0;
   DATA[30,20] := 148.808;
   DATA[30,21] := 156.1138;
   DATA[30,22] := 1.717361;
   DATA[30,23] := 946.2958;
   DATA[30,24] := 2.0;
   DATA[30,25] := 2.0;
   DATA[30,26] := 7.878621;
   DATA[30,27] := 144.9116;
   DATA[30,28] := 264.5475;
   DATA[30,29] := 12.11228;
   DATA[30,30] := 1.72725;
   DATA[30,31] := 1.278724;
   DATA[30,32] := 0.7348846;
   DATA[30,33] := 0.3065689;
   DATA[30,34] := 2.0;
   DATA[30,35] := 251.0414;
   DATA[30,36] := 1.649953;
   DATA[30,37] := 189.8071;
   DATA[30,38] := 0.000128152;
   DATA[30,39] := 1.0;
   DATA[31,0] := 2.598725;
   DATA[31,1] := 524.3383;
   DATA[31,2] := 2.0;
   DATA[31,3] := 2.0;
   DATA[31,4] := 262.0161;
   DATA[31,5] := 8.390669;
   DATA[31,6] := 328.6337;
   DATA[31,7] := 2.439881;
   DATA[31,8] := 2.0;
   DATA[31,9] := 2.0;
   DATA[31,10] := 2.0;
   DATA[31,11] := 19.68756;
   DATA[31,12] := 2.212215;
   DATA[31,13] := 957.3667;
   DATA[31,14] := 1.0;
   DATA[31,15] := 2.0;
   DATA[31,16] := 1.0;
   DATA[31,17] := 1.0;
   DATA[31,18] := 1.0;
   DATA[31,19] := 2.0;
   DATA[31,20] := 148.808;
   DATA[31,21] := 156.1138;
   DATA[31,22] := 1.717489;
   DATA[31,23] := 946.4881;
   DATA[31,24] := 2.0;
   DATA[31,25] := 2.0;
   DATA[31,26] := 7.878621;
   DATA[31,27] := 144.9116;
   DATA[31,28] := 264.5475;
   DATA[31,29] := 12.11228;
   DATA[31,30] := 1.72725;
   DATA[31,31] := 1.299603;
   DATA[31,32] := 0.7348846;
   DATA[31,33] := 0.3065689;
   DATA[31,34] := 2.0;
   DATA[31,35] := 251.0414;
   DATA[31,36] := 1.649953;
   DATA[31,37] := 189.8071;
   DATA[31,38] := 0.000128152;
   DATA[31,39] := 1.0;
   DATA[32,0] := 2.639721;
   DATA[32,1] := 524.5346;
   DATA[32,2] := 2.0;
   DATA[32,3] := 2.0;
   DATA[32,4] := 262.0161;
   DATA[32,5] := 8.390669;
   DATA[32,6] := 328.4799;
   DATA[32,7] := 2.439881;
   DATA[32,8] := 2.0;
   DATA[32,9] := 2.0;
   DATA[32,10] := 2.0;
   DATA[32,11] := 19.68756;
   DATA[32,12] := 2.212215;
   DATA[32,13] := 957.7673;
   DATA[32,14] := 1.0;
   DATA[32,15] := 2.0;
   DATA[32,16] := 1.0;
   DATA[32,17] := 1.0;
   DATA[32,18] := 1.0;
   DATA[32,19] := 2.0;
   DATA[32,20] := 148.808;
   DATA[32,21] := 156.1138;
   DATA[32,22] := 1.717874;
   DATA[32,23] := 946.2189;
   DATA[32,24] := 2.0;
   DATA[32,25] := 2.0;
   DATA[32,26] := 7.878621;
   DATA[32,27] := 144.9116;
   DATA[32,28] := 264.5475;
   DATA[32,29] := 12.11228;
   DATA[32,30] := 1.72725;
   DATA[32,31] := 1.302293;
   DATA[32,32] := 0.7348846;
   DATA[32,33] := 0.3075937;
   DATA[32,34] := 2.0;
   DATA[32,35] := 251.0414;
   DATA[32,36] := 1.649953;
   DATA[32,37] := 189.8071;
   DATA[32,38] := 0.000128152;
   DATA[32,39] := 1.0;
   DATA[33,0] := 2.667585;
   DATA[33,1] := 524.2991;
   DATA[33,2] := 2.0;
   DATA[33,3] := 2.0;
   DATA[33,4] := 262.0161;
   DATA[33,5] := 8.392271;
   DATA[33,6] := 328.403;
   DATA[33,7] := 2.439881;
   DATA[33,8] := 2.0;
   DATA[33,9] := 2.0;
   DATA[33,10] := 2.0;
   DATA[33,11] := 19.68756;
   DATA[33,12] := 2.212215;
   DATA[33,13] := 957.4869;
   DATA[33,14] := 1.0;
   DATA[33,15] := 2.0;
   DATA[33,16] := 1.0;
   DATA[33,17] := 1.0;
   DATA[33,18] := 1.0;
   DATA[33,19] := 2.0;
   DATA[33,20] := 148.808;
   DATA[33,21] := 155.96;
   DATA[33,22] := 1.717874;
   DATA[33,23] := 946.3343;
   DATA[33,24] := 2.0;
   DATA[33,25] := 2.0;
   DATA[33,26] := 7.878621;
   DATA[33,27] := 144.9116;
   DATA[33,28] := 264.5475;
   DATA[33,29] := 12.11228;
   DATA[33,30] := 1.725711;
   DATA[33,31] := 1.292814;
   DATA[33,32] := 0.7348846;
   DATA[33,33] := 0.3069532;
   DATA[33,34] := 2.0;
   DATA[33,35] := 250.9453;
   DATA[33,36] := 1.649953;
   DATA[33,37] := 189.5988;
   DATA[33,38] := 0.000128152;
   DATA[33,39] := 1.0;
   DATA[34,0] := 2.673029;
   DATA[34,1] := 524.2991;
   DATA[34,2] := 2.0;
   DATA[34,3] := 2.0;
   DATA[34,4] := 262.0161;
   DATA[34,5] := 8.392271;
   DATA[34,6] := 328.403;
   DATA[34,7] := 2.439881;
   DATA[34,8] := 2.0;
   DATA[34,9] := 2.0;
   DATA[34,10] := 2.0;
   DATA[34,11] := 19.68756;
   DATA[34,12] := 2.212215;
   DATA[34,13] := 957.7272;
   DATA[34,14] := 1.0;
   DATA[34,15] := 2.0;
   DATA[34,16] := 1.0;
   DATA[34,17] := 1.0;
   DATA[34,18] := 1.0;
   DATA[34,19] := 2.0;
   DATA[34,20] := 148.808;
   DATA[34,21] := 155.96;
   DATA[34,22] := 1.717874;
   DATA[34,23] := 946.2574;
   DATA[34,24] := 2.0;
   DATA[34,25] := 2.0;
   DATA[34,26] := 7.878621;
   DATA[34,27] := 144.9116;
   DATA[34,28] := 264.5475;
   DATA[34,29] := 12.11228;
   DATA[34,30] := 1.72507;
   DATA[34,31] := 1.283592;
   DATA[34,32] := 0.7348846;
   DATA[34,33] := 0.3068251;
   DATA[34,34] := 2.0;
   DATA[34,35] := 250.8171;
   DATA[34,36] := 1.649953;
   DATA[34,37] := 189.5988;
   DATA[34,38] := 0.000128152;
   DATA[34,39] := 1.0;
   DATA[35,0] := 2.653172;
   DATA[35,1] := 524.2206;
   DATA[35,2] := 2.0;
   DATA[35,3] := 2.0;
   DATA[35,4] := 262.0161;
   DATA[35,5] := 8.392271;
   DATA[35,6] := 328.403;
   DATA[35,7] := 2.439881;
   DATA[35,8] := 2.0;
   DATA[35,9] := 2.0;
   DATA[35,10] := 2.0;
   DATA[35,11] := 19.74838;
   DATA[35,12] := 2.209909;
   DATA[35,13] := 958.0076;
   DATA[35,14] := 1.0;
   DATA[35,15] := 2.0;
   DATA[35,16] := 1.0;
   DATA[35,17] := 1.0;
   DATA[35,18] := 1.0;
   DATA[35,19] := 2.0;
   DATA[35,20] := 148.808;
   DATA[35,21] := 155.96;
   DATA[35,22] := 1.71608;
   DATA[35,23] := 946.4112;
   DATA[35,24] := 2.0;
   DATA[35,25] := 2.0;
   DATA[35,26] := 7.878621;
   DATA[35,27] := 144.9116;
   DATA[35,28] := 264.5475;
   DATA[35,29] := 12.11228;
   DATA[35,30] := 1.72507;
   DATA[35,31] := 1.274625;
   DATA[35,32] := 0.7348846;
   DATA[35,33] := 0.3068251;
   DATA[35,34] := 2.0;
   DATA[35,35] := 250.7049;
   DATA[35,36] := 1.649953;
   DATA[35,37] := 189.5828;
   DATA[35,38] := 0.000128152;
   DATA[35,39] := 1.0;
   DATA[36,0] := 2.629152;
   DATA[36,1] := 524.4561;
   DATA[36,2] := 2.0;
   DATA[36,3] := 2.0;
   DATA[36,4] := 262.0161;
   DATA[36,5] := 8.392271;
   DATA[36,6] := 328.403;
   DATA[36,7] := 2.439881;
   DATA[36,8] := 2.0;
   DATA[36,9] := 2.0;
   DATA[36,10] := 2.0;
   DATA[36,11] := 19.74838;
   DATA[36,12] := 2.209653;
   DATA[36,13] := 958.288;
   DATA[36,14] := 1.0;
   DATA[36,15] := 2.0;
   DATA[36,16] := 1.0;
   DATA[36,17] := 1.0;
   DATA[36,18] := 1.0;
   DATA[36,19] := 2.0;
   DATA[36,20] := 148.808;
   DATA[36,21] := 155.96;
   DATA[36,22] := 1.71608;
   DATA[36,23] := 946.2189;
   DATA[36,24] := 2.0;
   DATA[36,25] := 2.0;
   DATA[36,26] := 7.878621;
   DATA[36,27] := 144.9116;
   DATA[36,28] := 264.5475;
   DATA[36,29] := 12.11228;
   DATA[36,30] := 1.726737;
   DATA[36,31] := 1.271679;
   DATA[36,32] := 0.7348846;
   DATA[36,33] := 0.3068251;
   DATA[36,34] := 2.0;
   DATA[36,35] := 250.7049;
   DATA[36,36] := 1.649953;
   DATA[36,37] := 189.4546;
   DATA[36,38] := 0.000128152;
   DATA[36,39] := 1.0;
   DATA[37,0] := 2.622105;
   DATA[37,1] := 524.4561;
   DATA[37,2] := 2.0;
   DATA[37,3] := 2.0;
   DATA[37,4] := 262.0161;
   DATA[37,5] := 8.392271;
   DATA[37,6] := 328.403;
   DATA[37,7] := 2.439881;
   DATA[37,8] := 2.0;
   DATA[37,9] := 2.0;
   DATA[37,10] := 2.0;
   DATA[37,11] := 19.74838;
   DATA[37,12] := 2.209653;
   DATA[37,13] := 958.2078;
   DATA[37,14] := 1.0;
   DATA[37,15] := 2.0;
   DATA[37,16] := 1.0;
   DATA[37,17] := 1.0;
   DATA[37,18] := 1.0;
   DATA[37,19] := 2.0;
   DATA[37,20] := 148.808;
   DATA[37,21] := 155.96;
   DATA[37,22] := 1.71608;
   DATA[37,23] := 946.1036;
   DATA[37,24] := 2.0;
   DATA[37,25] := 2.0;
   DATA[37,26] := 7.878621;
   DATA[37,27] := 144.9116;
   DATA[37,28] := 264.5475;
   DATA[37,29] := 12.11228;
   DATA[37,30] := 1.726737;
   DATA[37,31] := 1.271679;
   DATA[37,32] := 0.7359089;
   DATA[37,33] := 0.3083624;
   DATA[37,34] := 2.0;
   DATA[37,35] := 250.7049;
   DATA[37,36] := 1.649953;
   DATA[37,37] := 189.4546;
   DATA[37,38] := 0.000128152;
   DATA[37,39] := 1.0;
   DATA[38,0] := 2.619543;
   DATA[38,1] := 524.8486;
   DATA[38,2] := 2.0;
   DATA[38,3] := 2.0;
   DATA[38,4] := 262.0161;
   DATA[38,5] := 8.392271;
   DATA[38,6] := 328.403;
   DATA[38,7] := 2.439881;
   DATA[38,8] := 2.0;
   DATA[38,9] := 2.0;
   DATA[38,10] := 2.0;
   DATA[38,11] := 19.74838;
   DATA[38,12] := 2.209653;
   DATA[38,13] := 958.4882;
   DATA[38,14] := 1.0;
   DATA[38,15] := 2.0;
   DATA[38,16] := 1.0;
   DATA[38,17] := 1.0;
   DATA[38,18] := 1.0;
   DATA[38,19] := 2.0;
   DATA[38,20] := 148.808;
   DATA[38,21] := 155.96;
   DATA[38,22] := 1.711723;
   DATA[38,23] := 946.1036;
   DATA[38,24] := 2.0;
   DATA[38,25] := 2.0;
   DATA[38,26] := 7.878621;
   DATA[38,27] := 144.9116;
   DATA[38,28] := 264.5475;
   DATA[38,29] := 12.11228;
   DATA[38,30] := 1.724045;
   DATA[38,31] := 1.281286;
   DATA[38,32] := 0.7359089;
   DATA[38,33] := 0.3084265;
   DATA[38,34] := 2.0;
   DATA[38,35] := 250.7049;
   DATA[38,36] := 1.649953;
   DATA[38,37] := 189.4226;
   DATA[38,38] := 0.000128152;
   DATA[38,39] := 1.0;
   DATA[39,0] := 2.606412;
   DATA[39,1] := 525.3982;
   DATA[39,2] := 2.0;
   DATA[39,3] := 2.0;
   DATA[39,4] := 262.0161;
   DATA[39,5] := 8.392271;
   DATA[39,6] := 328.403;
   DATA[39,7] := 2.439881;
   DATA[39,8] := 2.0;
   DATA[39,9] := 2.0;
   DATA[39,10] := 2.0;
   DATA[39,11] := 19.68436;
   DATA[39,12] := 2.209653;
   DATA[39,13] := 958.328;
   DATA[39,14] := 1.0;
   DATA[39,15] := 2.0;
   DATA[39,16] := 1.0;
   DATA[39,17] := 1.0;
   DATA[39,18] := 1.0;
   DATA[39,19] := 2.0;
   DATA[39,20] := 148.808;
   DATA[39,21] := 155.96;
   DATA[39,22] := 1.711466;
   DATA[39,23] := 946.4112;
   DATA[39,24] := 2.0;
   DATA[39,25] := 2.0;
   DATA[39,26] := 7.878621;
   DATA[39,27] := 144.9116;
   DATA[39,28] := 264.5475;
   DATA[39,29] := 12.11228;
   DATA[39,30] := 1.724045;
   DATA[39,31] := 1.289612;
   DATA[39,32] := 0.7359089;
   DATA[39,33] := 0.3084265;
   DATA[39,34] := 2.0;
   DATA[39,35] := 250.7049;
   DATA[39,36] := 1.649953;
   DATA[39,37] := 189.3425;
   DATA[39,38] := 0.000128152;
   DATA[39,39] := 1.0;
   DATA[40,0] := 2.589117;
   DATA[40,1] := 525.3196;
   DATA[40,2] := 2.0;
   DATA[40,3] := 2.0;
   DATA[40,4] := 262.0161;
   DATA[40,5] := 8.392271;
   DATA[40,6] := 328.403;
   DATA[40,7] := 2.439881;
   DATA[40,8] := 2.0;
   DATA[40,9] := 2.0;
   DATA[40,10] := 2.0;
   DATA[40,11] := 19.65555;
   DATA[40,12] := 2.209653;
   DATA[40,13] := 958.6084;
   DATA[40,14] := 1.0;
   DATA[40,15] := 2.0;
   DATA[40,16] := 1.0;
   DATA[40,17] := 1.0;
   DATA[40,18] := 1.0;
   DATA[40,19] := 2.0;
   DATA[40,20] := 148.808;
   DATA[40,21] := 155.96;
   DATA[40,22] := 1.711466;
   DATA[40,23] := 946.6419;
   DATA[40,24] := 2.0;
   DATA[40,25] := 2.0;
   DATA[40,26] := 7.878621;
   DATA[40,27] := 144.9116;
   DATA[40,28] := 264.5475;
   DATA[40,29] := 12.45834;
   DATA[40,30] := 1.724045;
   DATA[40,31] := 1.292046;
   DATA[40,32] := 0.7359089;
   DATA[40,33] := 0.3084265;
   DATA[40,34] := 2.0;
   DATA[40,35] := 250.6569;
   DATA[40,36] := 1.649953;
   DATA[40,37] := 189.3425;
   DATA[40,38] := 0.000128152;
   DATA[40,39] := 1.0;
   DATA[41,0] := 2.574704;
   DATA[41,1] := 525.5159;
   DATA[41,2] := 2.0;
   DATA[41,3] := 2.0;
   DATA[41,4] := 262.0161;
   DATA[41,5] := 8.39131;
   DATA[41,6] := 328.403;
   DATA[41,7] := 2.439881;
   DATA[41,8] := 2.0;
   DATA[41,9] := 2.0;
   DATA[41,10] := 2.0;
   DATA[41,11] := 19.62994;
   DATA[41,12] := 2.209653;
   DATA[41,13] := 958.9689;
   DATA[41,14] := 1.0;
   DATA[41,15] := 2.0;
   DATA[41,16] := 1.0;
   DATA[41,17] := 1.0;
   DATA[41,18] := 1.0;
   DATA[41,19] := 2.0;
   DATA[41,20] := 148.808;
   DATA[41,21] := 155.96;
   DATA[41,22] := 1.711466;
   DATA[41,23] := 946.3343;
   DATA[41,24] := 2.0;
   DATA[41,25] := 2.0;
   DATA[41,26] := 7.878621;
   DATA[41,27] := 144.9116;
   DATA[41,28] := 264.5475;
   DATA[41,29] := 12.45834;
   DATA[41,30] := 1.724045;
   DATA[41,31] := 1.292046;
   DATA[41,32] := 0.7359089;
   DATA[41,33] := 0.3084265;
   DATA[41,34] := 2.0;
   DATA[41,35] := 250.5447;
   DATA[41,36] := 1.649953;
   DATA[41,37] := 189.3425;
   DATA[41,38] := 0.000128152;
   DATA[41,39] := 1.0;
   DATA[42,0] := 2.556129;
   DATA[42,1] := 525.6729;
   DATA[42,2] := 2.0;
   DATA[42,3] := 2.0;
   DATA[42,4] := 262.0161;
   DATA[42,5] := 8.389067;
   DATA[42,6] := 328.403;
   DATA[42,7] := 2.439881;
   DATA[42,8] := 2.0;
   DATA[42,9] := 2.0;
   DATA[42,10] := 2.0;
   DATA[42,11] := 19.62033;
   DATA[42,12] := 2.209653;
   DATA[42,13] := 959.0891;
   DATA[42,14] := 1.0;
   DATA[42,15] := 2.0;
   DATA[42,16] := 1.0;
   DATA[42,17] := 1.0;
   DATA[42,18] := 1.0;
   DATA[42,19] := 2.0;
   DATA[42,20] := 148.808;
   DATA[42,21] := 155.96;
   DATA[42,22] := 1.711466;
   DATA[42,23] := 946.3343;
   DATA[42,24] := 2.0;
   DATA[42,25] := 2.0;
   DATA[42,26] := 7.878621;
   DATA[42,27] := 144.9116;
   DATA[42,28] := 264.5475;
   DATA[42,29] := 12.45834;
   DATA[42,30] := 1.724045;
   DATA[42,31] := 1.287947;
   DATA[42,32] := 0.7355248;
   DATA[42,33] := 0.3084265;
   DATA[42,34] := 2.0;
   DATA[42,35] := 250.5447;
   DATA[42,36] := 1.649953;
   DATA[42,37] := 189.3425;
   DATA[42,38] := 0.000128152;
   DATA[42,39] := 1.0;
   DATA[43,0] := 2.545559;
   DATA[43,1] := 525.9084;
   DATA[43,2] := 2.0;
   DATA[43,3] := 2.0;
   DATA[43,4] := 262.0161;
   DATA[43,5] := 8.389067;
   DATA[43,6] := 328.403;
   DATA[43,7] := 2.437318;
   DATA[43,8] := 2.0;
   DATA[43,9] := 2.0;
   DATA[43,10] := 2.0;
   DATA[43,11] := 19.62033;
   DATA[43,12] := 2.209653;
   DATA[43,13] := 959.1691;
   DATA[43,14] := 1.0;
   DATA[43,15] := 2.0;
   DATA[43,16] := 1.0;
   DATA[43,17] := 1.0;
   DATA[43,18] := 1.0;
   DATA[43,19] := 2.0;
   DATA[43,20] := 148.808;
   DATA[43,21] := 155.96;
   DATA[43,22] := 1.711466;
   DATA[43,23] := 946.4112;
   DATA[43,24] := 2.0;
   DATA[43,25] := 2.0;
   DATA[43,26] := 7.878621;
   DATA[43,27] := 144.9116;
   DATA[43,28] := 264.5475;
   DATA[43,29] := 12.22763;
   DATA[43,30] := 1.723789;
   DATA[43,31] := 1.272192;
   DATA[43,32] := 0.7348846;
   DATA[43,33] := 0.3084265;
   DATA[43,34] := 2.0;
   DATA[43,35] := 250.5447;
   DATA[43,36] := 1.649953;
   DATA[43,37] := 189.3425;
   DATA[43,38] := 0.000128152;
   DATA[43,39] := 1.0;
   DATA[44,0] := 2.524741;
   DATA[44,1] := 525.7907;
   DATA[44,2] := 2.0;
   DATA[44,3] := 2.0;
   DATA[44,4] := 262.0161;
   DATA[44,5] := 8.389067;
   DATA[44,6] := 328.403;
   DATA[44,7] := 2.437318;
   DATA[44,8] := 2.0;
   DATA[44,9] := 2.0;
   DATA[44,10] := 2.0;
   DATA[44,11] := 19.67796;
   DATA[44,12] := 2.209653;
   DATA[44,13] := 959.4095;
   DATA[44,14] := 1.0;
   DATA[44,15] := 2.0;
   DATA[44,16] := 1.0;
   DATA[44,17] := 1.0;
   DATA[44,18] := 1.0;
   DATA[44,19] := 2.0;
   DATA[44,20] := 148.808;
   DATA[44,21] := 155.96;
   DATA[44,22] := 1.710826;
   DATA[44,23] := 946.5266;
   DATA[44,24] := 2.0;
   DATA[44,25] := 2.0;
   DATA[44,26] := 7.878621;
   DATA[44,27] := 145.091;
   DATA[44,28] := 264.5475;
   DATA[44,29] := 12.22763;
   DATA[44,30] := 1.722123;
   DATA[44,31] := 1.271295;
   DATA[44,32] := 0.7348846;
   DATA[44,33] := 0.3084265;
   DATA[44,34] := 2.0;
   DATA[44,35] := 250.5447;
   DATA[44,36] := 1.649953;
   DATA[44,37] := 189.3745;
   DATA[44,38] := 0.000128152;
   DATA[44,39] := 1.0;
   DATA[45,0] := 2.512891;
   DATA[45,1] := 525.9084;
   DATA[45,2] := 2.0;
   DATA[45,3] := 2.0;
   DATA[45,4] := 262.0161;
   DATA[45,5] := 8.389067;
   DATA[45,6] := 328.403;
   DATA[45,7] := 2.437318;
   DATA[45,8] := 2.0;
   DATA[45,9] := 2.0;
   DATA[45,10] := 2.0;
   DATA[45,11] := 19.67796;
   DATA[45,12] := 2.210678;
   DATA[45,13] := 959.4896;
   DATA[45,14] := 1.0;
   DATA[45,15] := 2.0;
   DATA[45,16] := 1.0;
   DATA[45,17] := 1.0;
   DATA[45,18] := 1.0;
   DATA[45,19] := 2.0;
   DATA[45,20] := 148.808;
   DATA[45,21] := 155.96;
   DATA[45,22] := 1.710826;
   DATA[45,23] := 946.2574;
   DATA[45,24] := 2.0;
   DATA[45,25] := 2.0;
   DATA[45,26] := 7.878621;
   DATA[45,27] := 145.091;
   DATA[45,28] := 264.3873;
   DATA[45,29] := 12.22763;
   DATA[45,30] := 1.722123;
   DATA[45,31] := 1.270655;
   DATA[45,32] := 0.7348846;
   DATA[45,33] := 0.3064407;
   DATA[45,34] := 2.0;
   DATA[45,35] := 250.5447;
   DATA[45,36] := 1.649953;
   DATA[45,37] := 189.3745;
   DATA[45,38] := 0.000128152;
   DATA[45,39] := 1.0;
   DATA[46,0] := 2.495276;
   DATA[46,1] := 525.7122;
   DATA[46,2] := 2.0;
   DATA[46,3] := 2.0;
   DATA[46,4] := 262.0161;
   DATA[46,5] := 8.389067;
   DATA[46,6] := 328.4286;
   DATA[46,7] := 2.43924;
   DATA[46,8] := 2.0;
   DATA[46,9] := 2.0;
   DATA[46,10] := 2.0;
   DATA[46,11] := 19.67796;
   DATA[46,12] := 2.2126;
   DATA[46,13] := 959.8901;
   DATA[46,14] := 1.0;
   DATA[46,15] := 2.0;
   DATA[46,16] := 1.0;
   DATA[46,17] := 1.0;
   DATA[46,18] := 1.0;
   DATA[46,19] := 2.0;
   DATA[46,20] := 148.808;
   DATA[46,21] := 155.96;
   DATA[46,22] := 1.712363;
   DATA[46,23] := 946.2189;
   DATA[46,24] := 2.0;
   DATA[46,25] := 2.0;
   DATA[46,26] := 7.878621;
   DATA[46,27] := 145.091;
   DATA[46,28] := 264.3873;
   DATA[46,29] := 12.11228;
   DATA[46,30] := 1.722123;
   DATA[46,31] := 1.274753;
   DATA[46,32] := 0.7348846;
   DATA[46,33] := 0.3064407;
   DATA[46,34] := 2.0;
   DATA[46,35] := 250.721;
   DATA[46,36] := 1.649953;
   DATA[46,37] := 189.5347;
   DATA[46,38] := 0.000128152;
   DATA[46,39] := 1.0;
   DATA[47,0] := 2.480863;
   DATA[47,1] := 525.5944;
   DATA[47,2] := 2.0;
   DATA[47,3] := 2.0;
   DATA[47,4] := 262.0161;
   DATA[47,5] := 8.389067;
   DATA[47,6] := 328.5312;
   DATA[47,7] := 2.440393;
   DATA[47,8] := 2.0;
   DATA[47,9] := 2.0;
   DATA[47,10] := 2.0;
   DATA[47,11] := 19.62354;
   DATA[47,12] := 2.213496;
   DATA[47,13] := 959.8901;
   DATA[47,14] := 1.0;
   DATA[47,15] := 2.0;
   DATA[47,16] := 1.0;
   DATA[47,17] := 1.0;
   DATA[47,18] := 1.0;
   DATA[47,19] := 2.0;
   DATA[47,20] := 148.808;
   DATA[47,21] := 155.96;
   DATA[47,22] := 1.714542;
   DATA[47,23] := 946.4496;
   DATA[47,24] := 2.0;
   DATA[47,25] := 2.0;
   DATA[47,26] := 7.878621;
   DATA[47,27] := 145.091;
   DATA[47,28] := 264.3873;
   DATA[47,29] := 12.03538;
   DATA[47,30] := 1.722379;
   DATA[47,31] := 1.290765;
   DATA[47,32] := 0.7348846;
   DATA[47,33] := 0.3064407;
   DATA[47,34] := 2.0;
   DATA[47,35] := 250.8331;
   DATA[47,36] := 1.649953;
   DATA[47,37] := 189.5347;
   DATA[47,38] := 0.000128152;
   DATA[47,39] := 1.0;
   DATA[48,0] := 2.460366;
   DATA[48,1] := 525.3196;
   DATA[48,2] := 2.0;
   DATA[48,3] := 2.0;
   DATA[48,4] := 262.0161;
   DATA[48,5] := 8.389067;
   DATA[48,6] := 328.5312;
   DATA[48,7] := 2.440393;
   DATA[48,8] := 2.0;
   DATA[48,9] := 2.0;
   DATA[48,10] := 2.0;
   DATA[48,11] := 19.62354;
   DATA[48,12] := 2.213496;
   DATA[48,13] := 959.8901;
   DATA[48,14] := 1.0;
   DATA[48,15] := 2.0;
   DATA[48,16] := 1.0;
   DATA[48,17] := 1.0;
   DATA[48,18] := 1.0;
   DATA[48,19] := 2.0;
   DATA[48,20] := 148.808;
   DATA[48,21] := 155.96;
   DATA[48,22] := 1.714542;
   DATA[48,23] := 946.3343;
   DATA[48,24] := 2.0;
   DATA[48,25] := 2.0;
   DATA[48,26] := 7.878621;
   DATA[48,27] := 145.091;
   DATA[48,28] := 264.3873;
   DATA[48,29] := 12.03538;
   DATA[48,30] := 1.724173;
   DATA[48,31] := 1.307929;
   DATA[48,32] := 0.7348846;
   DATA[48,33] := 0.3064407;
   DATA[48,34] := 2.0;
   DATA[48,35] := 250.8812;
   DATA[48,36] := 1.649953;
   DATA[48,37] := 189.5347;
   DATA[48,38] := 0.000128152;
   DATA[48,39] := 1.0;
   DATA[49,0] := 2.448195;
   DATA[49,1] := 525.3982;
   DATA[49,2] := 2.0;
   DATA[49,3] := 2.0;
   DATA[49,4] := 262.0161;
   DATA[49,5] := 8.389067;
   DATA[49,6] := 328.5312;
   DATA[49,7] := 2.440393;
   DATA[49,8] := 2.0;
   DATA[49,9] := 2.0;
   DATA[49,10] := 2.0;
   DATA[49,11] := 19.63954;
   DATA[49,12] := 2.212856;
   DATA[49,13] := 959.6898;
   DATA[49,14] := 1.0;
   DATA[49,15] := 2.0;
   DATA[49,16] := 1.0;
   DATA[49,17] := 1.0;
   DATA[49,18] := 1.0;
   DATA[49,19] := 2.0;
   DATA[49,20] := 148.808;
   DATA[49,21] := 155.96;
   DATA[49,22] := 1.715183;
   DATA[49,23] := 946.2958;
   DATA[49,24] := 2.0;
   DATA[49,25] := 2.0;
   DATA[49,26] := 7.878621;
   DATA[49,27] := 145.091;
   DATA[49,28] := 264.3873;
   DATA[49,29] := 12.03538;
   DATA[49,30] := 1.726737;
   DATA[49,31] := 1.307801;
   DATA[49,32] := 0.7348846;
   DATA[49,33] := 0.3064407;
   DATA[49,34] := 2.0;
   DATA[49,35] := 250.9132;
   DATA[49,36] := 1.649953;
   DATA[49,37] := 189.6629;
   DATA[49,38] := 0.000128152;
   DATA[49,39] := 1.0;
   DATA[50,0] := 2.431221;
   DATA[50,1] := 525.5944;
   DATA[50,2] := 2.0;
   DATA[50,3] := 2.0;
   DATA[50,4] := 262.0161;
   DATA[50,5] := 8.389067;
   DATA[50,6] := 328.5312;
   DATA[50,7] := 2.440393;
   DATA[50,8] := 2.0;
   DATA[50,9] := 2.0;
   DATA[50,10] := 2.0;
   DATA[50,11] := 19.65235;
   DATA[50,12] := 2.212215;
   DATA[50,13] := 959.9702;
   DATA[50,14] := 1.0;
   DATA[50,15] := 2.0;
   DATA[50,16] := 1.0;
   DATA[50,17] := 1.0;
   DATA[50,18] := 1.0;
   DATA[50,19] := 2.0;
   DATA[50,20] := 148.808;
   DATA[50,21] := 155.96;
   DATA[50,22] := 1.715183;
   DATA[50,23] := 946.2189;
   DATA[50,24] := 2.0;
   DATA[50,25] := 2.0;
   DATA[50,26] := 7.878621;
   DATA[50,27] := 145.091;
   DATA[50,28] := 264.3873;
   DATA[50,29] := 12.03538;
   DATA[50,30] := 1.726737;
   DATA[50,31] := 1.306136;
   DATA[50,32] := 0.7348846;
   DATA[50,33] := 0.3064407;
   DATA[50,34] := 2.0;
   DATA[50,35] := 250.9933;
   DATA[50,36] := 1.649953;
   DATA[50,37] := 189.759;
   DATA[50,38] := 0.000128152;
   DATA[50,39] := 1.0;
   DATA[51,0] := 2.420331;
   DATA[51,1] := 525.5944;
   DATA[51,2] := 2.0;
   DATA[51,3] := 2.0;
   DATA[51,4] := 262.0161;
   DATA[51,5] := 8.391951;
   DATA[51,6] := 328.5312;
   DATA[51,7] := 2.441675;
   DATA[51,8] := 2.0;
   DATA[51,9] := 2.0;
   DATA[51,10] := 2.0;
   DATA[51,11] := 19.65235;
   DATA[51,12] := 2.210678;
   DATA[51,13] := 959.81;
   DATA[51,14] := 1.0;
   DATA[51,15] := 2.0;
   DATA[51,16] := 1.0;
   DATA[51,17] := 1.0;
   DATA[51,18] := 1.0;
   DATA[51,19] := 2.0;
   DATA[51,20] := 148.808;
   DATA[51,21] := 155.96;
   DATA[51,22] := 1.715183;
   DATA[51,23] := 946.4112;
   DATA[51,24] := 2.0;
   DATA[51,25] := 2.0;
   DATA[51,26] := 7.878621;
   DATA[51,27] := 144.7834;
   DATA[51,28] := 264.2912;
   DATA[51,29] := 12.03538;
   DATA[51,30] := 1.727634;
   DATA[51,31] := 1.307929;
   DATA[51,32] := 0.7348846;
   DATA[51,33] := 0.3064407;
   DATA[51,34] := 2.0;
   DATA[51,35] := 251.0574;
   DATA[51,36] := 1.649953;
   DATA[51,37] := 189.759;
   DATA[51,38] := 0.000128152;
   DATA[51,39] := 1.0;
   DATA[52,0] := 2.420331;
   DATA[52,1] := 525.3982;
   DATA[52,2] := 2.0;
   DATA[52,3] := 2.0;
   DATA[52,4] := 262.0161;
   DATA[52,5] := 8.391951;
   DATA[52,6] := 328.5312;
   DATA[52,7] := 2.441675;
   DATA[52,8] := 2.0;
   DATA[52,9] := 2.0;
   DATA[52,10] := 2.0;
   DATA[52,11] := 19.65235;
   DATA[52,12] := 2.210678;
   DATA[52,13] := 960.1304;
   DATA[52,14] := 1.0;
   DATA[52,15] := 2.0;
   DATA[52,16] := 1.0;
   DATA[52,17] := 1.0;
   DATA[52,18] := 1.0;
   DATA[52,19] := 2.0;
   DATA[52,20] := 148.808;
   DATA[52,21] := 155.96;
   DATA[52,22] := 1.716592;
   DATA[52,23] := 946.8342;
   DATA[52,24] := 2.0;
   DATA[52,25] := 2.0;
   DATA[52,26] := 7.878621;
   DATA[52,27] := 144.7834;
   DATA[52,28] := 264.2592;
   DATA[52,29] := 12.03538;
   DATA[52,30] := 1.728531;
   DATA[52,31] := 1.29243;
   DATA[52,32] := 0.7348846;
   DATA[52,33] := 0.3064407;
   DATA[52,34] := 2.0;
   DATA[52,35] := 251.0574;
   DATA[52,36] := 1.649953;
   DATA[52,37] := 189.759;
   DATA[52,38] := 0.000128152;
   DATA[52,39] := 1.0;
   DATA[53,0] := 2.435384;
   DATA[53,1] := 525.7122;
   DATA[53,2] := 2.0;
   DATA[53,3] := 2.0;
   DATA[53,4] := 262.0161;
   DATA[53,5] := 8.391951;
   DATA[53,6] := 328.5312;
   DATA[53,7] := 2.440906;
   DATA[53,8] := 2.0;
   DATA[53,9] := 2.0;
   DATA[53,10] := 2.0;
   DATA[53,11] := 19.65235;
   DATA[53,12] := 2.21055;
   DATA[53,13] := 960.1304;
   DATA[53,14] := 1.0;
   DATA[53,15] := 2.0;
   DATA[53,16] := 1.0;
   DATA[53,17] := 1.0;
   DATA[53,18] := 1.0;
   DATA[53,19] := 2.0;
   DATA[53,20] := 148.808;
   DATA[53,21] := 155.96;
   DATA[53,22] := 1.717233;
   DATA[53,23] := 946.9111;
   DATA[53,24] := 2.0;
   DATA[53,25] := 2.0;
   DATA[53,26] := 7.878621;
   DATA[53,27] := 145.0397;
   DATA[53,28] := 264.2592;
   DATA[53,29] := 12.03538;
   DATA[53,30] := 1.728531;
   DATA[53,31] := 1.28641;
   DATA[53,32] := 0.7348846;
   DATA[53,33] := 0.3064407;
   DATA[53,34] := 2.0;
   DATA[53,35] := 251.0574;
   DATA[53,36] := 1.649953;
   DATA[53,37] := 189.759;
   DATA[53,38] := 0.000128152;
   DATA[53,39] := 1.0;
   DATA[54,0] := 2.481504;
   DATA[54,1] := 525.6729;
   DATA[54,2] := 2.0;
   DATA[54,3] := 2.0;
   DATA[54,4] := 262.0161;
   DATA[54,5] := 8.391951;
   DATA[54,6] := 328.5312;
   DATA[54,7] := 2.440906;
   DATA[54,8] := 2.0;
   DATA[54,9] := 2.0;
   DATA[54,10] := 2.0;
   DATA[54,11] := 19.70357;
   DATA[54,12] := 2.209397;
   DATA[54,13] := 960.0103;
   DATA[54,14] := 1.0;
   DATA[54,15] := 2.0;
   DATA[54,16] := 1.0;
   DATA[54,17] := 1.0;
   DATA[54,18] := 1.0;
   DATA[54,19] := 2.0;
   DATA[54,20] := 148.808;
   DATA[54,21] := 155.96;
   DATA[54,22] := 1.717233;
   DATA[54,23] := 946.5266;
   DATA[54,24] := 2.0;
   DATA[54,25] := 2.0;
   DATA[54,26] := 7.878621;
   DATA[54,27] := 145.0397;
   DATA[54,28] := 264.2592;
   DATA[54,29] := 12.03538;
   DATA[54,30] := 1.728531;
   DATA[54,31] := 1.287434;
   DATA[54,32] := 0.7348846;
   DATA[54,33] := 0.3071454;
   DATA[54,34] := 2.0;
   DATA[54,35] := 251.0574;
   DATA[54,36] := 1.649953;
   DATA[54,37] := 189.759;
   DATA[54,38] := 0.000128152;
   DATA[54,39] := 1.0;
   DATA[55,0] := 2.519617;
   DATA[55,1] := 525.5944;
   DATA[55,2] := 2.0;
   DATA[55,3] := 2.0;
   DATA[55,4] := 262.0161;
   DATA[55,5] := 8.391951;
   DATA[55,6] := 328.5312;
   DATA[55,7] := 2.440906;
   DATA[55,8] := 2.0;
   DATA[55,9] := 2.0;
   DATA[55,10] := 2.0;
   DATA[55,11] := 19.70357;
   DATA[55,12] := 2.208884;
   DATA[55,13] := 960.1705;
   DATA[55,14] := 1.0;
   DATA[55,15] := 2.0;
   DATA[55,16] := 1.0;
   DATA[55,17] := 1.0;
   DATA[55,18] := 1.0;
   DATA[55,19] := 2.0;
   DATA[55,20] := 148.808;
   DATA[55,21] := 155.96;
   DATA[55,22] := 1.717233;
   DATA[55,23] := 946.4112;
   DATA[55,24] := 2.0;
   DATA[55,25] := 2.0;
   DATA[55,26] := 7.878621;
   DATA[55,27] := 145.0397;
   DATA[55,28] := 264.2592;
   DATA[55,29] := 12.03538;
   DATA[55,30] := 1.728531;
   DATA[55,31] := 1.280646;
   DATA[55,32] := 0.7348846;
   DATA[55,33] := 0.3071454;
   DATA[55,34] := 2.0;
   DATA[55,35] := 251.0574;
   DATA[55,36] := 1.649953;
   DATA[55,37] := 189.759;
   DATA[55,38] := 0.000128152;
   DATA[55,39] := 1.0;
   DATA[56,0] := 2.554847;
   DATA[56,1] := 525.5944;
   DATA[56,2] := 2.0;
   DATA[56,3] := 2.0;
   DATA[56,4] := 262.0161;
   DATA[56,5] := 8.391951;
   DATA[56,6] := 328.5312;
   DATA[56,7] := 2.440906;
   DATA[56,8] := 2.0;
   DATA[56,9] := 2.0;
   DATA[56,10] := 2.0;
   DATA[56,11] := 19.70357;
   DATA[56,12] := 2.208884;
   DATA[56,13] := 960.0904;
   DATA[56,14] := 1.0;
   DATA[56,15] := 2.0;
   DATA[56,16] := 1.0;
   DATA[56,17] := 1.0;
   DATA[56,18] := 1.0;
   DATA[56,19] := 2.0;
   DATA[56,20] := 148.808;
   DATA[56,21] := 155.96;
   DATA[56,22] := 1.718643;
   DATA[56,23] := 946.3343;
   DATA[56,24] := 2.0;
   DATA[56,25] := 2.0;
   DATA[56,26] := 7.878621;
   DATA[56,27] := 145.0397;
   DATA[56,28] := 264.2592;
   DATA[56,29] := 12.03538;
   DATA[56,30] := 1.726993;
   DATA[56,31] := 1.288075;
   DATA[56,32] := 0.7348846;
   DATA[56,33] := 0.3066329;
   DATA[56,34] := 2.0;
   DATA[56,35] := 251.0574;
   DATA[56,36] := 1.649953;
   DATA[56,37] := 189.759;
   DATA[56,38] := 0.000128152;
   DATA[56,39] := 1.0;
   DATA[57,0] := 2.602569;
   DATA[57,1] := 525.5159;
   DATA[57,2] := 2.0;
   DATA[57,3] := 2.0;
   DATA[57,4] := 262.0161;
   DATA[57,5] := 8.391951;
   DATA[57,6] := 328.5312;
   DATA[57,7] := 2.440906;
   DATA[57,8] := 2.0;
   DATA[57,9] := 2.0;
   DATA[57,10] := 2.0;
   DATA[57,11] := 19.75479;
   DATA[57,12] := 2.208884;
   DATA[57,13] := 959.81;
   DATA[57,14] := 1.0;
   DATA[57,15] := 2.0;
   DATA[57,16] := 1.0;
   DATA[57,17] := 1.0;
   DATA[57,18] := 1.0;
   DATA[57,19] := 2.0;
   DATA[57,20] := 148.808;
   DATA[57,21] := 155.96;
   DATA[57,22] := 1.719924;
   DATA[57,23] := 946.3343;
   DATA[57,24] := 2.0;
   DATA[57,25] := 2.0;
   DATA[57,26] := 7.878621;
   DATA[57,27] := 145.0397;
   DATA[57,28] := 264.2592;
   DATA[57,29] := 12.03538;
   DATA[57,30] := 1.726609;
   DATA[57,31] := 1.292046;
   DATA[57,32] := 0.7348846;
   DATA[57,33] := 0.3065689;
   DATA[57,34] := 2.0;
   DATA[57,35] := 251.0574;
   DATA[57,36] := 1.649953;
   DATA[57,37] := 189.759;
   DATA[57,38] := 0.000128152;
   DATA[57,39] := 1.0;
   DATA[58,0] := 2.632995;
   DATA[58,1] := 525.5159;
   DATA[58,2] := 2.0;
   DATA[58,3] := 2.0;
   DATA[58,4] := 262.0161;
   DATA[58,5] := 8.391951;
   DATA[58,6] := 328.5055;
   DATA[58,7] := 2.440906;
   DATA[58,8] := 2.0;
   DATA[58,9] := 2.0;
   DATA[58,10] := 2.0;
   DATA[58,11] := 19.75479;
   DATA[58,12] := 2.208884;
   DATA[58,13] := 959.6097;
   DATA[58,14] := 1.0;
   DATA[58,15] := 2.0;
   DATA[58,16] := 1.0;
   DATA[58,17] := 1.0;
   DATA[58,18] := 1.0;
   DATA[58,19] := 2.0;
   DATA[58,20] := 148.808;
   DATA[58,21] := 155.96;
   DATA[58,22] := 1.719924;
   DATA[58,23] := 946.3343;
   DATA[58,24] := 2.0;
   DATA[58,25] := 2.0;
   DATA[58,26] := 7.878621;
   DATA[58,27] := 145.0397;
   DATA[58,28] := 264.2592;
   DATA[58,29] := 12.03538;
   DATA[58,30] := 1.726609;
   DATA[58,31] := 1.285513;
   DATA[58,32] := 0.7348846;
   DATA[58,33] := 0.3065689;
   DATA[58,34] := 2.0;
   DATA[58,35] := 251.0734;
   DATA[58,36] := 1.649953;
   DATA[58,37] := 189.9673;
   DATA[58,38] := 0.000128152;
   DATA[58,39] := 1.0;
   DATA[59,0] := 2.649329;
   DATA[59,1] := 525.5944;
   DATA[59,2] := 2.0;
   DATA[59,3] := 2.0;
   DATA[59,4] := 262.0161;
   DATA[59,5] := 8.391951;
   DATA[59,6] := 328.5055;
   DATA[59,7] := 2.4427;
   DATA[59,8] := 2.0;
   DATA[59,9] := 2.0;
   DATA[59,10] := 2.0;
   DATA[59,11] := 19.70677;
   DATA[59,12] := 2.207347;
   DATA[59,13] := 959.7299;
   DATA[59,14] := 1.0;
   DATA[59,15] := 2.0;
   DATA[59,16] := 1.0;
   DATA[59,17] := 1.0;
   DATA[59,18] := 1.0;
   DATA[59,19] := 2.0;
   DATA[59,20] := 148.808;
   DATA[59,21] := 155.96;
   DATA[59,22] := 1.719924;
   DATA[59,23] := 946.1036;
   DATA[59,24] := 2.0;
   DATA[59,25] := 2.0;
   DATA[59,26] := 7.878621;
   DATA[59,27] := 145.0397;
   DATA[59,28] := 264.4194;
   DATA[59,29] := 12.03538;
   DATA[59,30] := 1.726609;
   DATA[59,31] := 1.272704;
   DATA[59,32] := 0.7348846;
   DATA[59,33] := 0.3065689;
   DATA[59,34] := 2.0;
   DATA[59,35] := 251.2337;
   DATA[59,36] := 1.649953;
   DATA[59,37] := 189.9673;
   DATA[59,38] := 0.000128152;
   DATA[59,39] := 1.0;
   DATA[60,0] := 2.656375;
   DATA[60,1] := 525.5159;
   DATA[60,2] := 2.0;
   DATA[60,3] := 2.0;
   DATA[60,4] := 262.0161;
   DATA[60,5] := 8.391951;
   DATA[60,6] := 328.403;
   DATA[60,7] := 2.443085;
   DATA[60,8] := 2.0;
   DATA[60,9] := 2.0;
   DATA[60,10] := 2.0;
   DATA[60,11] := 19.69076;
   DATA[60,12] := 2.20645;
   DATA[60,13] := 959.6898;
   DATA[60,14] := 1.0;
   DATA[60,15] := 2.0;
   DATA[60,16] := 1.0;
   DATA[60,17] := 1.0;
   DATA[60,18] := 1.0;
   DATA[60,19] := 2.0;
   DATA[60,20] := 148.808;
   DATA[60,21] := 155.96;
   DATA[60,22] := 1.719924;
   DATA[60,23] := 946.0651;
   DATA[60,24] := 2.0;
   DATA[60,25] := 2.0;
   DATA[60,26] := 7.878621;
   DATA[60,27] := 145.0397;
   DATA[60,28] := 264.4194;
   DATA[60,29] := 12.03538;
   DATA[60,30] := 1.728916;
   DATA[60,31] := 1.271679;
   DATA[60,32] := 0.7348846;
   DATA[60,33] := 0.3065689;
   DATA[60,34] := 2.0;
   DATA[60,35] := 251.2817;
   DATA[60,36] := 1.649953;
   DATA[60,37] := 189.9673;
   DATA[60,38] := 0.000128152;
   DATA[60,39] := 1.0;
   DATA[61,0] := 2.652211;
   DATA[61,1] := 525.1234;
   DATA[61,2] := 2.0;
   DATA[61,3] := 2.0;
   DATA[61,4] := 262.0161;
   DATA[61,5] := 8.391951;
   DATA[61,6] := 328.3517;
   DATA[61,7] := 2.443085;
   DATA[61,8] := 2.0;
   DATA[61,9] := 2.0;
   DATA[61,10] := 2.0;
   DATA[61,11] := 19.65235;
   DATA[61,12] := 2.20645;
   DATA[61,13] := 959.6898;
   DATA[61,14] := 1.0;
   DATA[61,15] := 2.0;
   DATA[61,16] := 1.0;
   DATA[61,17] := 1.0;
   DATA[61,18] := 1.0;
   DATA[61,19] := 2.0;
   DATA[61,20] := 148.808;
   DATA[61,21] := 155.96;
   DATA[61,22] := 1.719924;
   DATA[61,23] := 945.9498;
   DATA[61,24] := 2.0;
   DATA[61,25] := 2.0;
   DATA[61,26] := 7.878621;
   DATA[61,27] := 145.0397;
   DATA[61,28] := 264.4194;
   DATA[61,29] := 12.03538;
   DATA[61,30] := 1.729428;
   DATA[61,31] := 1.270911;
   DATA[61,32] := 0.7348846;
   DATA[61,33] := 0.3065689;
   DATA[61,34] := 2.0;
   DATA[61,35] := 251.3138;
   DATA[61,36] := 1.649953;
   DATA[61,37] := 190.1436;
   DATA[61,38] := 0.000128152;
   DATA[61,39] := 1.0;
   DATA[62,0] := 2.636838;
   DATA[62,1] := 525.2019;
   DATA[62,2] := 2.0;
   DATA[62,3] := 2.0;
   DATA[62,4] := 262.0161;
   DATA[62,5] := 8.389708;
   DATA[62,6] := 328.3517;
   DATA[62,7] := 2.441034;
   DATA[62,8] := 2.0;
   DATA[62,9] := 2.0;
   DATA[62,10] := 2.0;
   DATA[62,11] := 19.65235;
   DATA[62,12] := 2.20645;
   DATA[62,13] := 959.7299;
   DATA[62,14] := 1.0;
   DATA[62,15] := 2.0;
   DATA[62,16] := 1.0;
   DATA[62,17] := 1.0;
   DATA[62,18] := 1.0;
   DATA[62,19] := 2.0;
   DATA[62,20] := 148.808;
   DATA[62,21] := 155.96;
   DATA[62,22] := 1.719924;
   DATA[62,23] := 946.2958;
   DATA[62,24] := 2.0;
   DATA[62,25] := 2.0;
   DATA[62,26] := 7.878621;
   DATA[62,27] := 145.0397;
   DATA[62,28] := 264.4194;
   DATA[62,29] := 12.03538;
   DATA[62,30] := 1.73071;
   DATA[62,31] := 1.277699;
   DATA[62,32] := 0.7348846;
   DATA[62,33] := 0.3065689;
   DATA[62,34] := 2.0;
   DATA[62,35] := 251.506;
   DATA[62,36] := 1.649953;
   DATA[62,37] := 190.1436;
   DATA[62,38] := 0.000128152;
   DATA[62,39] := 1.0;
   DATA[63,0] := 2.625628;
   DATA[63,1] := 525.2411;
   DATA[63,2] := 2.0;
   DATA[63,3] := 2.0;
   DATA[63,4] := 262.0161;
   DATA[63,5] := 8.389708;
   DATA[63,6] := 328.3517;
   DATA[63,7] := 2.440137;
   DATA[63,8] := 2.0;
   DATA[63,9] := 2.0;
   DATA[63,10] := 2.0;
   DATA[63,11] := 19.70357;
   DATA[63,12] := 2.20645;
   DATA[63,13] := 959.5296;
   DATA[63,14] := 1.0;
   DATA[63,15] := 2.0;
   DATA[63,16] := 1.0;
   DATA[63,17] := 1.0;
   DATA[63,18] := 1.0;
   DATA[63,19] := 2.0;
   DATA[63,20] := 148.808;
   DATA[63,21] := 156.1907;
   DATA[63,22] := 1.719924;
   DATA[63,23] := 946.4881;
   DATA[63,24] := 2.0;
   DATA[63,25] := 2.0;
   DATA[63,26] := 7.878621;
   DATA[63,27] := 145.0397;
   DATA[63,28] := 264.4194;
   DATA[63,29] := 12.03538;
   DATA[63,30] := 1.731479;
   DATA[63,31] := 1.282311;
   DATA[63,32] := 0.7348846;
   DATA[63,33] := 0.3065689;
   DATA[63,34] := 2.0;
   DATA[63,35] := 251.506;
   DATA[63,36] := 1.649953;
   DATA[63,37] := 190.1436;
   DATA[63,38] := 0.000128152;
   DATA[63,39] := 1.0;
   DATA[64,0] := 2.620504;
   DATA[64,1] := 524.8094;
   DATA[64,2] := 2.0;
   DATA[64,3] := 2.0;
   DATA[64,4] := 262.0161;
   DATA[64,5] := 8.389708;
   DATA[64,6] := 328.3517;
   DATA[64,7] := 2.440137;
   DATA[64,8] := 2.0;
   DATA[64,9] := 2.0;
   DATA[64,10] := 2.0;
   DATA[64,11] := 19.74198;
   DATA[64,12] := 2.20645;
   DATA[64,13] := 959.6097;
   DATA[64,14] := 1.0;
   DATA[64,15] := 2.0;
   DATA[64,16] := 1.0;
   DATA[64,17] := 1.0;
   DATA[64,18] := 1.0;
   DATA[64,19] := 2.0;
   DATA[64,20] := 148.808;
   DATA[64,21] := 156.1907;
   DATA[64,22] := 1.720693;
   DATA[64,23] := 946.6419;
   DATA[64,24] := 2.0;
   DATA[64,25] := 2.0;
   DATA[64,26] := 7.878621;
   DATA[64,27] := 145.0397;
   DATA[64,28] := 264.4194;
   DATA[64,29] := 12.30454;
   DATA[64,30] := 1.731479;
   DATA[64,31] := 1.282311;
   DATA[64,32] := 0.7348846;
   DATA[64,33] := 0.3065689;
   DATA[64,34] := 2.0;
   DATA[64,35] := 251.506;
   DATA[64,36] := 1.649953;
   DATA[64,37] := 190.1436;
   DATA[64,38] := 0.000128152;
   DATA[64,39] := 1.0;
   DATA[65,0] := 2.610575;
   DATA[65,1] := 524.4561;
   DATA[65,2] := 2.0;
   DATA[65,3] := 2.0;
   DATA[65,4] := 262.0161;
   DATA[65,5] := 8.389708;
   DATA[65,6] := 328.3517;
   DATA[65,7] := 2.440521;
   DATA[65,8] := 2.0;
   DATA[65,9] := 2.0;
   DATA[65,10] := 2.0;
   DATA[65,11] := 19.69076;
   DATA[65,12] := 2.20645;
   DATA[65,13] := 959.3293;
   DATA[65,14] := 1.0;
   DATA[65,15] := 2.0;
   DATA[65,16] := 1.0;
   DATA[65,17] := 1.0;
   DATA[65,18] := 1.0;
   DATA[65,19] := 2.0;
   DATA[65,20] := 148.808;
   DATA[65,21] := 156.1907;
   DATA[65,22] := 1.720693;
   DATA[65,23] := 946.9111;
   DATA[65,24] := 2.0;
   DATA[65,25] := 2.0;
   DATA[65,26] := 7.878621;
   DATA[65,27] := 145.0397;
   DATA[65,28] := 264.4194;
   DATA[65,29] := 12.30454;
   DATA[65,30] := 1.731479;
   DATA[65,31] := 1.282311;
   DATA[65,32] := 0.7348846;
   DATA[65,33] := 0.3065689;
   DATA[65,34] := 2.0;
   DATA[65,35] := 251.506;
   DATA[65,36] := 1.649953;
   DATA[65,37] := 190.1436;
   DATA[65,38] := 0.000128152;
   DATA[65,39] := 1.0;
   DATA[66,0] := 2.595202;
   DATA[66,1] := 524.0243;
   DATA[66,2] := 2.0;
   DATA[66,3] := 2.0;
   DATA[66,4] := 262.0161;
   DATA[66,5] := 8.389708;
   DATA[66,6] := 328.3517;
   DATA[66,7] := 2.441419;
   DATA[66,8] := 2.0;
   DATA[66,9] := 2.0;
   DATA[66,10] := 2.0;
   DATA[66,11] := 19.67476;
   DATA[66,12] := 2.209525;
   DATA[66,13] := 959.3694;
   DATA[66,14] := 1.0;
   DATA[66,15] := 2.0;
   DATA[66,16] := 1.0;
   DATA[66,17] := 1.0;
   DATA[66,18] := 1.0;
   DATA[66,19] := 2.0;
   DATA[66,20] := 148.808;
   DATA[66,21] := 156.0882;
   DATA[66,22] := 1.718643;
   DATA[66,23] := 946.988;
   DATA[66,24] := 2.0;
   DATA[66,25] := 2.0;
   DATA[66,26] := 7.878621;
   DATA[66,27] := 145.0397;
   DATA[66,28] := 264.4194;
   DATA[66,29] := 12.30454;
   DATA[66,30] := 1.732504;
   DATA[66,31] := 1.291405;
   DATA[66,32] := 0.7348846;
   DATA[66,33] := 0.3065689;
   DATA[66,34] := 2.0;
   DATA[66,35] := 251.506;
   DATA[66,36] := 1.649953;
   DATA[66,37] := 190.1436;
   DATA[66,38] := 0.000128152;
   DATA[66,39] := 1.0;
   DATA[67,0] := 2.575345;
   DATA[67,1] := 523.9458;
   DATA[67,2] := 2.0;
   DATA[67,3] := 2.0;
   DATA[67,4] := 262.0161;
   DATA[67,5] := 8.389708;
   DATA[67,6] := 328.3517;
   DATA[67,7] := 2.441419;
   DATA[67,8] := 2.0;
   DATA[67,9] := 2.0;
   DATA[67,10] := 2.0;
   DATA[67,11] := 19.67476;
   DATA[67,12] := 2.210166;
   DATA[67,13] := 959.5697;
   DATA[67,14] := 1.0;
   DATA[67,15] := 2.0;
   DATA[67,16] := 1.0;
   DATA[67,17] := 1.0;
   DATA[67,18] := 1.0;
   DATA[67,19] := 2.0;
   DATA[67,20] := 148.808;
   DATA[67,21] := 155.96;
   DATA[67,22] := 1.718643;
   DATA[67,23] := 947.2571;
   DATA[67,24] := 2.0;
   DATA[67,25] := 2.0;
   DATA[67,26] := 7.878621;
   DATA[67,27] := 145.0397;
   DATA[67,28] := 264.4194;
   DATA[67,29] := 12.30454;
   DATA[67,30] := 1.732504;
   DATA[67,31] := 1.29243;
   DATA[67,32] := 0.7348846;
   DATA[67,33] := 0.3065689;
   DATA[67,34] := 2.0;
   DATA[67,35] := 251.506;
   DATA[67,36] := 1.649953;
   DATA[67,37] := 190.1436;
   DATA[67,38] := 0.000128152;
   DATA[67,39] := 1.0;
   DATA[68,0] := 2.561253;
   DATA[68,1] := 523.8281;
   DATA[68,2] := 2.0;
   DATA[68,3] := 2.0;
   DATA[68,4] := 262.0161;
   DATA[68,5] := 8.391951;
   DATA[68,6] := 328.3517;
   DATA[68,7] := 2.441419;
   DATA[68,8] := 2.0;
   DATA[68,9] := 2.0;
   DATA[68,10] := 2.0;
   DATA[68,11] := 19.67476;
   DATA[68,12] := 2.212856;
   DATA[68,13] := 959.6898;
   DATA[68,14] := 1.0;
   DATA[68,15] := 2.0;
   DATA[68,16] := 1.0;
   DATA[68,17] := 1.0;
   DATA[68,18] := 1.0;
   DATA[68,19] := 2.0;
   DATA[68,20] := 148.808;
   DATA[68,21] := 155.96;
   DATA[68,22] := 1.718643;
   DATA[68,23] := 947.2571;
   DATA[68,24] := 2.0;
   DATA[68,25] := 2.0;
   DATA[68,26] := 7.878621;
   DATA[68,27] := 145.0397;
   DATA[68,28] := 264.4194;
   DATA[68,29] := 12.03538;
   DATA[68,30] := 1.732504;
   DATA[68,31] := 1.285129;
   DATA[68,32] := 0.7348846;
   DATA[68,33] := 0.3065689;
   DATA[68,34] := 2.0;
   DATA[68,35] := 251.506;
   DATA[68,36] := 1.649953;
   DATA[68,37] := 190.1436;
   DATA[68,38] := 0.000128152;
   DATA[68,39] := 1.0;
   DATA[69,0] := 2.561253;
   DATA[69,1] := 523.8281;
   DATA[69,2] := 2.0;
   DATA[69,3] := 2.0;
   DATA[69,4] := 262.0161;
   DATA[69,5] := 8.391951;
   DATA[69,6] := 328.3517;
   DATA[69,7] := 2.441419;
   DATA[69,8] := 2.0;
   DATA[69,9] := 2.0;
   DATA[69,10] := 2.0;
   DATA[69,11] := 19.67476;
   DATA[69,12] := 2.212856;
   DATA[69,13] := 959.6898;
   DATA[69,14] := 1.0;
   DATA[69,15] := 2.0;
   DATA[69,16] := 1.0;
   DATA[69,17] := 1.0;
   DATA[69,18] := 1.0;
   DATA[69,19] := 2.0;
   DATA[69,20] := 148.808;
   DATA[69,21] := 155.96;
   DATA[69,22] := 1.718643;
   DATA[69,23] := 947.2571;
   DATA[69,24] := 2.0;
   DATA[69,25] := 2.0;
   DATA[69,26] := 7.878621;
   DATA[69,27] := 145.0397;
   DATA[69,28] := 264.4194;
   DATA[69,29] := 12.03538;
   DATA[69,30] := 1.732504;
   DATA[69,31] := 1.285129;
   DATA[69,32] := 0.7348846;
   DATA[69,33] := 0.3065689;
   DATA[69,34] := 2.0;
   DATA[69,35] := 251.506;
   DATA[69,36] := 1.649953;
   DATA[69,37] := 190.1436;
   DATA[69,38] := 0.000128152;
   DATA[69,39] := 1.0;
   DATA[70,0] := 2.542677;
   DATA[70,1] := 524.1421;
   DATA[70,2] := 2.0;
   DATA[70,3] := 2.0;
   DATA[70,4] := 262.0161;
   DATA[70,5] := 8.391951;
   DATA[70,6] := 328.5568;
   DATA[70,7] := 2.441419;
   DATA[70,8] := 2.0;
   DATA[70,9] := 2.0;
   DATA[70,10] := 2.0;
   DATA[70,11] := 19.67476;
   DATA[70,12] := 2.212856;
   DATA[70,13] := 959.5697;
   DATA[70,14] := 1.0;
   DATA[70,15] := 2.0;
   DATA[70,16] := 1.0;
   DATA[70,17] := 1.0;
   DATA[70,18] := 1.0;
   DATA[70,19] := 2.0;
   DATA[70,20] := 148.808;
   DATA[70,21] := 155.96;
   DATA[70,22] := 1.719796;
   DATA[70,23] := 947.6031;
   DATA[70,24] := 2.0;
   DATA[70,25] := 2.0;
   DATA[70,26] := 7.878621;
   DATA[70,27] := 145.0397;
   DATA[70,28] := 264.4194;
   DATA[70,29] := 12.03538;
   DATA[70,30] := 1.731735;
   DATA[70,31] := 1.288587;
   DATA[70,32] := 0.7348846;
   DATA[70,33] := 0.3065689;
   DATA[70,34] := 2.0;
   DATA[70,35] := 251.506;
   DATA[70,36] := 1.649953;
   DATA[70,37] := 190.1436;
   DATA[70,38] := 0.000128152;
   DATA[70,39] := 1.0;
   DATA[71,0] := 2.528905;
   DATA[71,1] := 524.3383;
   DATA[71,2] := 2.0;
   DATA[71,3] := 2.0;
   DATA[71,4] := 262.0161;
   DATA[71,5] := 8.391951;
   DATA[71,6] := 328.5568;
   DATA[71,7] := 2.441419;
   DATA[71,8] := 2.0;
   DATA[71,9] := 2.0;
   DATA[71,10] := 2.0;
   DATA[71,11] := 19.61073;
   DATA[71,12] := 2.212856;
   DATA[71,13] := 959.9702;
   DATA[71,14] := 1.0;
   DATA[71,15] := 2.0;
   DATA[71,16] := 1.0;
   DATA[71,17] := 1.0;
   DATA[71,18] := 1.0;
   DATA[71,19] := 2.0;
   DATA[71,20] := 148.808;
   DATA[71,21] := 156.2164;
   DATA[71,22] := 1.720309;
   DATA[71,23] := 947.6801;
   DATA[71,24] := 2.0;
   DATA[71,25] := 2.0;
   DATA[71,26] := 7.878621;
   DATA[71,27] := 145.0397;
   DATA[71,28] := 264.4194;
   DATA[71,29] := 12.03538;
   DATA[71,30] := 1.731095;
   DATA[71,31] := 1.286666;
   DATA[71,32] := 0.7348846;
   DATA[71,33] := 0.3065689;
   DATA[71,34] := 2.0;
   DATA[71,35] := 251.506;
   DATA[71,36] := 1.665972;
   DATA[71,37] := 190.1436;
   DATA[71,38] := 0.000128152;
   DATA[71,39] := 1.0;
   DATA[72,0] := 2.51193;
   DATA[72,1] := 524.6131;
   DATA[72,2] := 2.0;
   DATA[72,3] := 2.0;
   DATA[72,4] := 262.0161;
   DATA[72,5] := 8.391951;
   DATA[72,6] := 328.5568;
   DATA[72,7] := 2.442828;
   DATA[72,8] := 2.0;
   DATA[72,9] := 2.0;
   DATA[72,10] := 2.0;
   DATA[72,11] := 19.57552;
   DATA[72,12] := 2.211318;
   DATA[72,13] := 960.1705;
   DATA[72,14] := 1.0;
   DATA[72,15] := 2.0;
   DATA[72,16] := 1.0;
   DATA[72,17] := 1.0;
   DATA[72,18] := 1.0;
   DATA[72,19] := 2.0;
   DATA[72,20] := 148.808;
   DATA[72,21] := 156.242;
   DATA[72,22] := 1.720309;
   DATA[72,23] := 947.5647;
   DATA[72,24] := 2.0;
   DATA[72,25] := 2.0;
   DATA[72,26] := 7.878621;
   DATA[72,27] := 145.0397;
   DATA[72,28] := 264.4194;
   DATA[72,29] := 12.03538;
   DATA[72,30] := 1.731095;
   DATA[72,31] := 1.288075;
   DATA[72,32] := 0.7348846;
   DATA[72,33] := 0.3065689;
   DATA[72,34] := 2.0;
   DATA[72,35] := 251.506;
   DATA[72,36] := 1.665972;
   DATA[72,37] := 190.1436;
   DATA[72,38] := 0.000128152;
   DATA[72,39] := 1.0;
   DATA[73,0] := 2.497518;
   DATA[73,1] := 524.6916;
   DATA[73,2] := 2.0;
   DATA[73,3] := 2.0;
   DATA[73,4] := 262.0161;
   DATA[73,5] := 8.391951;
   DATA[73,6] := 328.5568;
   DATA[73,7] := 2.442828;
   DATA[73,8] := 2.0;
   DATA[73,9] := 2.0;
   DATA[73,10] := 2.0;
   DATA[73,11] := 19.55631;
   DATA[73,12] := 2.21055;
   DATA[73,13] := 959.9702;
   DATA[73,14] := 1.0;
   DATA[73,15] := 2.0;
   DATA[73,16] := 1.0;
   DATA[73,17] := 1.0;
   DATA[73,18] := 1.0;
   DATA[73,19] := 2.0;
   DATA[73,20] := 148.808;
   DATA[73,21] := 156.242;
   DATA[73,22] := 1.720309;
   DATA[73,23] := 947.5647;
   DATA[73,24] := 2.0;
   DATA[73,25] := 2.0;
   DATA[73,26] := 7.878621;
   DATA[73,27] := 145.0397;
   DATA[73,28] := 264.4194;
   DATA[73,29] := 12.03538;
   DATA[73,30] := 1.731095;
   DATA[73,31] := 1.291533;
   DATA[73,32] := 0.7348846;
   DATA[73,33] := 0.3065689;
   DATA[73,34] := 2.0;
   DATA[73,35] := 251.506;
   DATA[73,36] := 1.665972;
   DATA[73,37] := 190.1436;
   DATA[73,38] := 0.000128152;
   DATA[73,39] := 1.0;
   DATA[74,0] := 2.473817;
   DATA[74,1] := 524.4561;
   DATA[74,2] := 2.0;
   DATA[74,3] := 2.0;
   DATA[74,4] := 262.0161;
   DATA[74,5] := 8.391951;
   DATA[74,6] := 328.5568;
   DATA[74,7] := 2.440137;
   DATA[74,8] := 2.0;
   DATA[74,9] := 2.0;
   DATA[74,10] := 2.0;
   DATA[74,11] := 19.55631;
   DATA[74,12] := 2.21055;
   DATA[74,13] := 960.1705;
   DATA[74,14] := 1.0;
   DATA[74,15] := 2.0;
   DATA[74,16] := 1.0;
   DATA[74,17] := 1.0;
   DATA[74,18] := 1.0;
   DATA[74,19] := 2.0;
   DATA[74,20] := 148.808;
   DATA[74,21] := 156.242;
   DATA[74,22] := 1.720309;
   DATA[74,23] := 947.8723;
   DATA[74,24] := 2.0;
   DATA[74,25] := 2.0;
   DATA[74,26] := 7.878621;
   DATA[74,27] := 145.0397;
   DATA[74,28] := 264.4194;
   DATA[74,29] := 12.03538;
   DATA[74,30] := 1.731095;
   DATA[74,31] := 1.291533;
   DATA[74,32] := 0.7355248;
   DATA[74,33] := 0.3065689;
   DATA[74,34] := 2.0;
   DATA[74,35] := 251.506;
   DATA[74,36] := 1.665972;
   DATA[74,37] := 190.1436;
   DATA[74,38] := 0.000128152;
   DATA[74,39] := 1.0;
   DATA[75,0] := 2.463248;
   DATA[75,1] := 524.7309;
   DATA[75,2] := 2.0;
   DATA[75,3] := 2.0;
   DATA[75,4] := 262.0161;
   DATA[75,5] := 8.391951;
   DATA[75,6] := 328.4286;
   DATA[75,7] := 2.440137;
   DATA[75,8] := 2.0;
   DATA[75,9] := 2.0;
   DATA[75,10] := 2.0;
   DATA[75,11] := 19.59472;
   DATA[75,12] := 2.21055;
   DATA[75,13] := 960.3307;
   DATA[75,14] := 1.0;
   DATA[75,15] := 2.0;
   DATA[75,16] := 1.0;
   DATA[75,17] := 1.0;
   DATA[75,18] := 1.0;
   DATA[75,19] := 2.0;
   DATA[75,20] := 148.808;
   DATA[75,21] := 156.242;
   DATA[75,22] := 1.720309;
   DATA[75,23] := 947.757;
   DATA[75,24] := 2.0;
   DATA[75,25] := 2.0;
   DATA[75,26] := 7.878621;
   DATA[75,27] := 145.0397;
   DATA[75,28] := 264.4194;
   DATA[75,29] := 12.03538;
   DATA[75,30] := 1.729428;
   DATA[75,31] := 1.291533;
   DATA[75,32] := 0.736421;
   DATA[75,33] := 0.3065689;
   DATA[75,34] := 2.0;
   DATA[75,35] := 251.2657;
   DATA[75,36] := 1.665972;
   DATA[75,37] := 189.9833;
   DATA[75,38] := 0.000128152;
   DATA[75,39] := 1.0;
   DATA[76,0] := 2.44179;
   DATA[76,1] := 524.6916;
   DATA[76,2] := 2.0;
   DATA[76,3] := 2.0;
   DATA[76,4] := 262.0161;
   DATA[76,5] := 8.391951;
   DATA[76,6] := 328.4286;
   DATA[76,7] := 2.440137;
   DATA[76,8] := 2.0;
   DATA[76,9] := 2.0;
   DATA[76,10] := 2.0;
   DATA[76,11] := 19.62354;
   DATA[76,12] := 2.21055;
   DATA[76,13] := 959.9702;
   DATA[76,14] := 1.0;
   DATA[76,15] := 2.0;
   DATA[76,16] := 1.0;
   DATA[76,17] := 1.0;
   DATA[76,18] := 1.0;
   DATA[76,19] := 2.0;
   DATA[76,20] := 148.808;
   DATA[76,21] := 156.242;
   DATA[76,22] := 1.719796;
   DATA[76,23] := 948.2184;
   DATA[76,24] := 2.0;
   DATA[76,25] := 2.0;
   DATA[76,26] := 7.878621;
   DATA[76,27] := 145.0397;
   DATA[76,28] := 264.4194;
   DATA[76,29] := 12.03538;
   DATA[76,30] := 1.726096;
   DATA[76,31] := 1.303446;
   DATA[76,32] := 0.736421;
   DATA[76,33] := 0.3065689;
   DATA[76,34] := 2.0;
   DATA[76,35] := 251.2657;
   DATA[76,36] := 1.665972;
   DATA[76,37] := 189.9833;
   DATA[76,38] := 0.000128152;
   DATA[76,39] := 1.0;
   DATA[77,0] := 2.431221;
   DATA[77,1] := 525.0842;
   DATA[77,2] := 2.0;
   DATA[77,3] := 2.0;
   DATA[77,4] := 262.0161;
   DATA[77,5] := 8.391951;
   DATA[77,6] := 328.4286;
   DATA[77,7] := 2.440137;
   DATA[77,8] := 2.0;
   DATA[77,9] := 2.0;
   DATA[77,10] := 2.0;
   DATA[77,11] := 19.64274;
   DATA[77,12] := 2.21055;
   DATA[77,13] := 960.0103;
   DATA[77,14] := 1.0;
   DATA[77,15] := 2.0;
   DATA[77,16] := 1.0;
   DATA[77,17] := 1.0;
   DATA[77,18] := 1.0;
   DATA[77,19] := 2.0;
   DATA[77,20] := 148.808;
   DATA[77,21] := 156.242;
   DATA[77,22] := 1.718515;
   DATA[77,23] := 948.6029;
   DATA[77,24] := 2.0;
   DATA[77,25] := 2.0;
   DATA[77,26] := 7.878621;
   DATA[77,27] := 145.0397;
   DATA[77,28] := 264.4194;
   DATA[77,29] := 12.03538;
   DATA[77,30] := 1.726096;
   DATA[77,31] := 1.311387;
   DATA[77,32] := 0.736421;
   DATA[77,33] := 0.3068891;
   DATA[77,34] := 2.0;
   DATA[77,35] := 250.9933;
   DATA[77,36] := 1.665972;
   DATA[77,37] := 189.8071;
   DATA[77,38] := 0.000128152;
   DATA[77,39] := 1.0;
   DATA[78,0] := 2.421932;
   DATA[78,1] := 525.2411;
   DATA[78,2] := 2.0;
   DATA[78,3] := 2.0;
   DATA[78,4] := 262.0161;
   DATA[78,5] := 8.391951;
   DATA[78,6] := 328.4286;
   DATA[78,7] := 2.440137;
   DATA[78,8] := 2.0;
   DATA[78,9] := 2.0;
   DATA[78,10] := 2.0;
   DATA[78,11] := 19.64274;
   DATA[78,12] := 2.208756;
   DATA[78,13] := 960.1304;
   DATA[78,14] := 1.0;
   DATA[78,15] := 2.0;
   DATA[78,16] := 1.0;
   DATA[78,17] := 1.0;
   DATA[78,18] := 1.0;
   DATA[78,19] := 2.0;
   DATA[78,20] := 148.808;
   DATA[78,21] := 156.242;
   DATA[78,22] := 1.718515;
   DATA[78,23] := 948.5645;
   DATA[78,24] := 2.0;
   DATA[78,25] := 2.0;
   DATA[78,26] := 7.878621;
   DATA[78,27] := 145.0397;
   DATA[78,28] := 264.2912;
   DATA[78,29] := 12.03538;
   DATA[78,30] := 1.725968;
   DATA[78,31] := 1.306008;
   DATA[78,32] := 0.736421;
   DATA[78,33] := 0.3068891;
   DATA[78,34] := 2.0;
   DATA[78,35] := 250.9933;
   DATA[78,36] := 1.665972;
   DATA[78,37] := 189.6629;
   DATA[78,38] := 0.000128152;
   DATA[78,39] := 1.0;
   DATA[79,0] := 2.420011;
   DATA[79,1] := 525.5159;
   DATA[79,2] := 2.0;
   DATA[79,3] := 2.0;
   DATA[79,4] := 262.0161;
   DATA[79,5] := 8.391951;
   DATA[79,6] := 328.4286;
   DATA[79,7] := 2.440137;
   DATA[79,8] := 2.0;
   DATA[79,9] := 2.0;
   DATA[79,10] := 2.0;
   DATA[79,11] := 19.64274;
   DATA[79,12] := 2.208756;
   DATA[79,13] := 959.9702;
   DATA[79,14] := 1.0;
   DATA[79,15] := 2.0;
   DATA[79,16] := 1.0;
   DATA[79,17] := 1.0;
   DATA[79,18] := 1.0;
   DATA[79,19] := 2.0;
   DATA[79,20] := 148.808;
   DATA[79,21] := 156.242;
   DATA[79,22] := 1.720309;
   DATA[79,23] := 948.7952;
   DATA[79,24] := 2.0;
   DATA[79,25] := 2.0;
   DATA[79,26] := 7.878621;
   DATA[79,27] := 145.1679;
   DATA[79,28] := 264.2912;
   DATA[79,29] := 12.03538;
   DATA[79,30] := 1.724814;
   DATA[79,31] := 1.306904;
   DATA[79,32] := 0.7353967;
   DATA[79,33] := 0.3068891;
   DATA[79,34] := 2.0;
   DATA[79,35] := 250.9933;
   DATA[79,36] := 1.665972;
   DATA[79,37] := 189.6629;
   DATA[79,38] := 0.000128152;
   DATA[79,39] := 1.0;
   DATA[80,0] := 2.447875;
   DATA[80,1] := 525.3196;
   DATA[80,2] := 2.0;
   DATA[80,3] := 2.0;
   DATA[80,4] := 262.0161;
   DATA[80,5] := 8.394835;
   DATA[80,6] := 328.4286;
   DATA[80,7] := 2.440137;
   DATA[80,8] := 2.0;
   DATA[80,9] := 2.0;
   DATA[80,10] := 2.0;
   DATA[80,11] := 19.65555;
   DATA[80,12] := 2.208756;
   DATA[80,13] := 960.3708;
   DATA[80,14] := 1.0;
   DATA[80,15] := 2.0;
   DATA[80,16] := 1.0;
   DATA[80,17] := 1.0;
   DATA[80,18] := 1.0;
   DATA[80,19] := 2.0;
   DATA[80,20] := 148.808;
   DATA[80,21] := 156.242;
   DATA[80,22] := 1.720309;
   DATA[80,23] := 948.9105;
   DATA[80,24] := 2.0;
   DATA[80,25] := 2.0;
   DATA[80,26] := 7.878621;
   DATA[80,27] := 145.2448;
   DATA[80,28] := 264.2912;
   DATA[80,29] := 12.03538;
   DATA[80,30] := 1.724814;
   DATA[80,31] := 1.297938;
   DATA[80,32] := 0.7353967;
   DATA[80,33] := 0.3068891;
   DATA[80,34] := 2.0;
   DATA[80,35] := 250.9933;
   DATA[80,36] := 1.665972;
   DATA[80,37] := 189.6629;
   DATA[80,38] := 0.000128152;
   DATA[80,39] := 1.0;
   DATA[81,0] := 2.500721;
   DATA[81,1] := 526.0262;
   DATA[81,2] := 2.0;
   DATA[81,3] := 2.0;
   DATA[81,4] := 262.0161;
   DATA[81,5] := 8.394835;
   DATA[81,6] := 328.4286;
   DATA[81,7] := 2.440137;
   DATA[81,8] := 2.0;
   DATA[81,9] := 2.0;
   DATA[81,10] := 2.0;
   DATA[81,11] := 19.65555;
   DATA[81,12] := 2.208756;
   DATA[81,13] := 960.2506;
   DATA[81,14] := 1.0;
   DATA[81,15] := 2.0;
   DATA[81,16] := 1.0;
   DATA[81,17] := 1.0;
   DATA[81,18] := 1.0;
   DATA[81,19] := 2.0;
   DATA[81,20] := 148.808;
   DATA[81,21] := 156.242;
   DATA[81,22] := 1.720309;
   DATA[81,23] := 949.1028;
   DATA[81,24] := 2.0;
   DATA[81,25] := 2.0;
   DATA[81,26] := 7.878621;
   DATA[81,27] := 145.2448;
   DATA[81,28] := 264.2592;
   DATA[81,29] := 12.03538;
   DATA[81,30] := 1.724814;
   DATA[81,31] := 1.292174;
   DATA[81,32] := 0.7353967;
   DATA[81,33] := 0.3066329;
   DATA[81,34] := 2.0;
   DATA[81,35] := 250.9933;
   DATA[81,36] := 1.569859;
   DATA[81,37] := 189.6629;
   DATA[81,38] := 0.000128152;
   DATA[81,39] := 1.0;
   DATA[82,0] := 2.543958;
   DATA[82,1] := 526.4973;
   DATA[82,2] := 2.0;
   DATA[82,3] := 2.0;
   DATA[82,4] := 262.0161;
   DATA[82,5] := 8.394835;
   DATA[82,6] := 328.4286;
   DATA[82,7] := 2.440137;
   DATA[82,8] := 2.0;
   DATA[82,9] := 2.0;
   DATA[82,10] := 2.0;
   DATA[82,11] := 19.65555;
   DATA[82,12] := 2.208756;
   DATA[82,13] := 960.0904;
   DATA[82,14] := 1.0;
   DATA[82,15] := 2.0;
   DATA[82,16] := 1.0;
   DATA[82,17] := 1.0;
   DATA[82,18] := 1.0;
   DATA[82,19] := 2.0;
   DATA[82,20] := 148.808;
   DATA[82,21] := 156.242;
   DATA[82,22] := 1.718643;
   DATA[82,23] := 949.1797;
   DATA[82,24] := 2.0;
   DATA[82,25] := 2.0;
   DATA[82,26] := 7.878621;
   DATA[82,27] := 145.2448;
   DATA[82,28] := 264.2592;
   DATA[82,29] := 12.03538;
   DATA[82,30] := 1.724814;
   DATA[82,31] := 1.288971;
   DATA[82,32] := 0.7353967;
   DATA[82,33] := 0.3065048;
   DATA[82,34] := 2.0;
   DATA[82,35] := 250.9933;
   DATA[82,36] := 1.569859;
   DATA[82,37] := 189.6629;
   DATA[82,38] := 0.000128152;
   DATA[82,39] := 1.0;
   DATA[83,0] := 2.570861;
   DATA[83,1] := 526.8898;
   DATA[83,2] := 2.0;
   DATA[83,3] := 2.0;
   DATA[83,4] := 262.0161;
   DATA[83,5] := 8.394835;
   DATA[83,6] := 328.4286;
   DATA[83,7] := 2.441034;
   DATA[83,8] := 2.0;
   DATA[83,9] := 2.0;
   DATA[83,10] := 2.0;
   DATA[83,11] := 19.65555;
   DATA[83,12] := 2.208756;
   DATA[83,13] := 959.8901;
   DATA[83,14] := 1.0;
   DATA[83,15] := 2.0;
   DATA[83,16] := 1.0;
   DATA[83,17] := 1.0;
   DATA[83,18] := 1.0;
   DATA[83,19] := 2.0;
   DATA[83,20] := 148.808;
   DATA[83,21] := 156.242;
   DATA[83,22] := 1.718643;
   DATA[83,23] := 949.2181;
   DATA[83,24] := 2.0;
   DATA[83,25] := 2.0;
   DATA[83,26] := 7.878621;
   DATA[83,27] := 145.2448;
   DATA[83,28] := 264.2592;
   DATA[83,29] := 12.03538;
   DATA[83,30] := 1.724814;
   DATA[83,31] := 1.282311;
   DATA[83,32] := 0.7353967;
   DATA[83,33] := 0.3065048;
   DATA[83,34] := 2.0;
   DATA[83,35] := 250.9933;
   DATA[83,36] := 1.569859;
   DATA[83,37] := 189.6629;
   DATA[83,38] := 0.000128152;
   DATA[83,39] := 1.0;
   DATA[84,0] := 2.614739;
   DATA[84,1] := 527.2038;
   DATA[84,2] := 2.0;
   DATA[84,3] := 2.0;
   DATA[84,4] := 262.0161;
   DATA[84,5] := 8.394835;
   DATA[84,6] := 328.4286;
   DATA[84,7] := 2.441034;
   DATA[84,8] := 2.0;
   DATA[84,9] := 2.0;
   DATA[84,10] := 2.0;
   DATA[84,11] := 19.65555;
   DATA[84,12] := 2.208756;
   DATA[84,13] := 959.8901;
   DATA[84,14] := 1.0;
   DATA[84,15] := 2.0;
   DATA[84,16] := 1.0;
   DATA[84,17] := 1.0;
   DATA[84,18] := 1.0;
   DATA[84,19] := 2.0;
   DATA[84,20] := 148.808;
   DATA[84,21] := 156.242;
   DATA[84,22] := 1.718643;
   DATA[84,23] := 949.8718;
   DATA[84,24] := 2.0;
   DATA[84,25] := 2.0;
   DATA[84,26] := 7.878621;
   DATA[84,27] := 145.1423;
   DATA[84,28] := 264.2592;
   DATA[84,29] := 12.03538;
   DATA[84,30] := 1.724814;
   DATA[84,31] := 1.27898;
   DATA[84,32] := 0.7353967;
   DATA[84,33] := 0.3065048;
   DATA[84,34] := 2.0;
   DATA[84,35] := 250.9933;
   DATA[84,36] := 1.569859;
   DATA[84,37] := 189.6629;
   DATA[84,38] := 0.000128152;
   DATA[84,39] := 1.0;
   DATA[85,0] := 2.645806;
   DATA[85,1] := 527.3608;
   DATA[85,2] := 2.0;
   DATA[85,3] := 2.0;
   DATA[85,4] := 262.2084;
   DATA[85,5] := 8.394835;
   DATA[85,6] := 328.4286;
   DATA[85,7] := 2.441034;
   DATA[85,8] := 2.0;
   DATA[85,9] := 2.0;
   DATA[85,10] := 2.0;
   DATA[85,11] := 19.65555;
   DATA[85,12] := 2.208756;
   DATA[85,13] := 960.0103;
   DATA[85,14] := 1.0;
   DATA[85,15] := 2.0;
   DATA[85,16] := 1.0;
   DATA[85,17] := 1.0;
   DATA[85,18] := 1.0;
   DATA[85,19] := 2.0;
   DATA[85,20] := 148.808;
   DATA[85,21] := 156.0882;
   DATA[85,22] := 1.720693;
   DATA[85,23] := 950.0641;
   DATA[85,24] := 2.0;
   DATA[85,25] := 2.0;
   DATA[85,26] := 7.878621;
   DATA[85,27] := 144.9885;
   DATA[85,28] := 264.2592;
   DATA[85,29] := 12.03538;
   DATA[85,30] := 1.724814;
   DATA[85,31] := 1.27232;
   DATA[85,32] := 0.7353967;
   DATA[85,33] := 0.3065048;
   DATA[85,34] := 2.0;
   DATA[85,35] := 250.9933;
   DATA[85,36] := 1.569859;
   DATA[85,37] := 189.7751;
   DATA[85,38] := 0.000128152;
   DATA[85,39] := 1.0;
   DATA[86,0] := 2.665023;
   DATA[86,1] := 527.4786;
   DATA[86,2] := 2.0;
   DATA[86,3] := 2.0;
   DATA[86,4] := 262.2084;
   DATA[86,5] := 8.394835;
   DATA[86,6] := 328.4286;
   DATA[86,7] := 2.441034;
   DATA[86,8] := 2.0;
   DATA[86,9] := 2.0;
   DATA[86,10] := 2.0;
   DATA[86,11] := 19.65555;
   DATA[86,12] := 2.208756;
   DATA[86,13] := 959.8901;
   DATA[86,14] := 1.0;
   DATA[86,15] := 2.0;
   DATA[86,16] := 1.0;
   DATA[86,17] := 1.0;
   DATA[86,18] := 1.0;
   DATA[86,19] := 2.0;
   DATA[86,20] := 148.808;
   DATA[86,21] := 156.0882;
   DATA[86,22] := 1.720693;
   DATA[86,23] := 950.1794;
   DATA[86,24] := 2.0;
   DATA[86,25] := 2.0;
   DATA[86,26] := 7.878621;
   DATA[86,27] := 144.9885;
   DATA[86,28] := 264.2592;
   DATA[86,29] := 12.03538;
   DATA[86,30] := 1.724814;
   DATA[86,31] := 1.270398;
   DATA[86,32] := 0.7353967;
   DATA[86,33] := 0.3065048;
   DATA[86,34] := 2.0;
   DATA[86,35] := 250.9933;
   DATA[86,36] := 1.569859;
   DATA[86,37] := 189.7751;
   DATA[86,38] := 0.000128152;
   DATA[86,39] := 1.0;
   DATA[87,0] := 2.666944;
   DATA[87,1] := 527.7534;
   DATA[87,2] := 2.0;
   DATA[87,3] := 2.0;
   DATA[87,4] := 262.2084;
   DATA[87,5] := 8.393553;
   DATA[87,6] := 328.4286;
   DATA[87,7] := 2.441547;
   DATA[87,8] := 2.0;
   DATA[87,9] := 2.0;
   DATA[87,10] := 2.0;
   DATA[87,11] := 19.65555;
   DATA[87,12] := 2.208756;
   DATA[87,13] := 959.5296;
   DATA[87,14] := 1.0;
   DATA[87,15] := 2.0;
   DATA[87,16] := 1.0;
   DATA[87,17] := 1.0;
   DATA[87,18] := 1.0;
   DATA[87,19] := 2.0;
   DATA[87,20] := 148.808;
   DATA[87,21] := 156.0882;
   DATA[87,22] := 1.720693;
   DATA[87,23] := 950.0641;
   DATA[87,24] := 2.0;
   DATA[87,25] := 2.0;
   DATA[87,26] := 7.878621;
   DATA[87,27] := 144.9885;
   DATA[87,28] := 264.2592;
   DATA[87,29] := 12.30454;
   DATA[87,30] := 1.724814;
   DATA[87,31] := 1.270398;
   DATA[87,32] := 0.7353967;
   DATA[87,33] := 0.3065048;
   DATA[87,34] := 2.0;
   DATA[87,35] := 250.9933;
   DATA[87,36] := 1.569859;
   DATA[87,37] := 189.7751;
   DATA[87,38] := 0.000128152;
   DATA[87,39] := 1.0;
   DATA[88,0] := 2.6394;
   DATA[88,1] := 528.2244;
   DATA[88,2] := 2.0;
   DATA[88,3] := 2.0;
   DATA[88,4] := 262.2084;
   DATA[88,5] := 8.391951;
   DATA[88,6] := 328.4286;
   DATA[88,7] := 2.443597;
   DATA[88,8] := 2.0;
   DATA[88,9] := 2.0;
   DATA[88,10] := 2.0;
   DATA[88,11] := 19.65555;
   DATA[88,12] := 2.209653;
   DATA[88,13] := 959.4896;
   DATA[88,14] := 1.0;
   DATA[88,15] := 2.0;
   DATA[88,16] := 1.0;
   DATA[88,17] := 1.0;
   DATA[88,18] := 1.0;
   DATA[88,19] := 2.0;
   DATA[88,20] := 148.808;
   DATA[88,21] := 156.0882;
   DATA[88,22] := 1.720693;
   DATA[88,23] := 950.2563;
   DATA[88,24] := 2.0;
   DATA[88,25] := 2.0;
   DATA[88,26] := 7.878621;
   DATA[88,27] := 144.9885;
   DATA[88,28] := 264.2592;
   DATA[88,29] := 12.30454;
   DATA[88,30] := 1.727378;
   DATA[88,31] := 1.284232;
   DATA[88,32] := 0.7353967;
   DATA[88,33] := 0.3065048;
   DATA[88,34] := 2.0;
   DATA[88,35] := 250.9933;
   DATA[88,36] := 1.569859;
   DATA[88,37] := 189.7751;
   DATA[88,38] := 0.000128152;
   DATA[88,39] := 1.0;
   DATA[89,0] := 2.620824;
   DATA[89,1] := 527.8711;
   DATA[89,2] := 2.0;
   DATA[89,3] := 2.0;
   DATA[89,4] := 261.9841;
   DATA[89,5] := 8.391951;
   DATA[89,6] := 328.4286;
   DATA[89,7] := 2.444751;
   DATA[89,8] := 2.0;
   DATA[89,9] := 2.0;
   DATA[89,10] := 2.0;
   DATA[89,11] := 19.60433;
   DATA[89,12] := 2.209653;
   DATA[89,13] := 959.5697;
   DATA[89,14] := 1.0;
   DATA[89,15] := 2.0;
   DATA[89,16] := 1.0;
   DATA[89,17] := 1.0;
   DATA[89,18] := 1.0;
   DATA[89,19] := 2.0;
   DATA[89,20] := 148.808;
   DATA[89,21] := 156.0882;
   DATA[89,22] := 1.719924;
   DATA[89,23] := 950.5255;
   DATA[89,24] := 2.0;
   DATA[89,25] := 2.0;
   DATA[89,26] := 7.878621;
   DATA[89,27] := 144.9885;
   DATA[89,28] := 264.2592;
   DATA[89,29] := 12.30454;
   DATA[89,30] := 1.727378;
   DATA[89,31] := 1.290765;
   DATA[89,32] := 0.7353967;
   DATA[89,33] := 0.3065048;
   DATA[89,34] := 2.0;
   DATA[89,35] := 250.9933;
   DATA[89,36] := 1.569859;
   DATA[89,37] := 189.7751;
   DATA[89,38] := 0.000128152;
   DATA[89,39] := 1.0;
   DATA[90,0] := 2.61634;
   DATA[90,1] := 528.0281;
   DATA[90,2] := 2.0;
   DATA[90,3] := 2.0;
   DATA[90,4] := 261.9841;
   DATA[90,5] := 8.391951;
   DATA[90,6] := 328.4286;
   DATA[90,7] := 2.444751;
   DATA[90,8] := 2.0;
   DATA[90,9] := 2.0;
   DATA[90,10] := 2.0;
   DATA[90,11] := 19.60433;
   DATA[90,12] := 2.209653;
   DATA[90,13] := 959.5697;
   DATA[90,14] := 1.0;
   DATA[90,15] := 2.0;
   DATA[90,16] := 1.0;
   DATA[90,17] := 1.0;
   DATA[90,18] := 1.0;
   DATA[90,19] := 2.0;
   DATA[90,20] := 148.808;
   DATA[90,21] := 156.0882;
   DATA[90,22] := 1.719284;
   DATA[90,23] := 950.6409;
   DATA[90,24] := 2.0;
   DATA[90,25] := 2.0;
   DATA[90,26] := 7.878621;
   DATA[90,27] := 145.1166;
   DATA[90,28] := 264.2592;
   DATA[90,29] := 12.30454;
   DATA[90,30] := 1.727378;
   DATA[90,31] := 1.285385;
   DATA[90,32] := 0.7353967;
   DATA[90,33] := 0.3065048;
   DATA[90,34] := 2.0;
   DATA[90,35] := 250.9933;
   DATA[90,36] := 1.681991;
   DATA[90,37] := 189.7751;
   DATA[90,38] := 0.000128152;
   DATA[90,39] := 1.0;
   DATA[91,0] := 2.61602;
   DATA[91,1] := 527.7534;
   DATA[91,2] := 2.0;
   DATA[91,3] := 2.0;
   DATA[91,4] := 261.9841;
   DATA[91,5] := 8.391951;
   DATA[91,6] := 328.4286;
   DATA[91,7] := 2.444751;
   DATA[91,8] := 2.0;
   DATA[91,9] := 2.0;
   DATA[91,10] := 2.0;
   DATA[91,11] := 19.60433;
   DATA[91,12] := 2.212215;
   DATA[91,13] := 959.4095;
   DATA[91,14] := 1.0;
   DATA[91,15] := 2.0;
   DATA[91,16] := 1.0;
   DATA[91,17] := 1.0;
   DATA[91,18] := 1.0;
   DATA[91,19] := 2.0;
   DATA[91,20] := 148.808;
   DATA[91,21] := 156.0882;
   DATA[91,22] := 1.719284;
   DATA[91,23] := 950.8331;
   DATA[91,24] := 2.0;
   DATA[91,25] := 2.0;
   DATA[91,26] := 7.878621;
   DATA[91,27] := 145.1679;
   DATA[91,28] := 264.2592;
   DATA[91,29] := 12.30454;
   DATA[91,30] := 1.727378;
   DATA[91,31] := 1.288843;
   DATA[91,32] := 0.7353967;
   DATA[91,33] := 0.3065048;
   DATA[91,34] := 2.0;
   DATA[91,35] := 250.9933;
   DATA[91,36] := 1.681991;
   DATA[91,37] := 189.7751;
   DATA[91,38] := 0.000128152;
   DATA[91,39] := 1.0;
   DATA[92,0] := 2.609294;
   DATA[92,1] := 527.4393;
   DATA[92,2] := 2.0;
   DATA[92,3] := 2.0;
   DATA[92,4] := 261.9841;
   DATA[92,5] := 8.391951;
   DATA[92,6] := 328.4286;
   DATA[92,7] := 2.443085;
   DATA[92,8] := 2.0;
   DATA[92,9] := 2.0;
   DATA[92,10] := 2.0;
   DATA[92,11] := 19.64274;
   DATA[92,12] := 2.212215;
   DATA[92,13] := 959.77;
   DATA[92,14] := 1.0;
   DATA[92,15] := 2.0;
   DATA[92,16] := 1.0;
   DATA[92,17] := 1.0;
   DATA[92,18] := 1.0;
   DATA[92,19] := 2.0;
   DATA[92,20] := 148.808;
   DATA[92,21] := 156.0882;
   DATA[92,22] := 1.718387;
   DATA[92,23] := 950.8716;
   DATA[92,24] := 2.0;
   DATA[92,25] := 2.0;
   DATA[92,26] := 7.878621;
   DATA[92,27] := 145.1679;
   DATA[92,28] := 264.2592;
   DATA[92,29] := 12.30454;
   DATA[92,30] := 1.727378;
   DATA[92,31] := 1.278468;
   DATA[92,32] := 0.7353967;
   DATA[92,33] := 0.3065048;
   DATA[92,34] := 2.0;
   DATA[92,35] := 250.9933;
   DATA[92,36] := 1.681991;
   DATA[92,37] := 189.7751;
   DATA[92,38] := 0.000128152;
   DATA[92,39] := 1.0;
   DATA[93,0] := 2.584313;
   DATA[93,1] := 527.2823;
   DATA[93,2] := 2.0;
   DATA[93,3] := 2.0;
   DATA[93,4] := 261.9841;
   DATA[93,5] := 8.391951;
   DATA[93,6] := 328.4286;
   DATA[93,7] := 2.442316;
   DATA[93,8] := 2.0;
   DATA[93,9] := 2.0;
   DATA[93,10] := 2.0;
   DATA[93,11] := 19.65875;
   DATA[93,12] := 2.212343;
   DATA[93,13] := 960.0904;
   DATA[93,14] := 1.0;
   DATA[93,15] := 2.0;
   DATA[93,16] := 1.0;
   DATA[93,17] := 1.0;
   DATA[93,18] := 1.0;
   DATA[93,19] := 2.0;
   DATA[93,20] := 148.808;
   DATA[93,21] := 156.0882;
   DATA[93,22] := 1.716849;
   DATA[93,23] := 951.0638;
   DATA[93,24] := 2.0;
   DATA[93,25] := 2.0;
   DATA[93,26] := 7.877019;
   DATA[93,27] := 145.1679;
   DATA[93,28] := 264.2592;
   DATA[93,29] := 12.30454;
   DATA[93,30] := 1.727378;
   DATA[93,31] := 1.263097;
   DATA[93,32] := 0.7353967;
   DATA[93,33] := 0.3065048;
   DATA[93,34] := 2.0;
   DATA[93,35] := 251.1055;
   DATA[93,36] := 1.649953;
   DATA[93,37] := 189.7751;
   DATA[93,38] := 0.000128152;
   DATA[93,39] := 1.0;
   DATA[94,0] := 2.572463;
   DATA[94,1] := 527.2823;
   DATA[94,2] := 2.0;
   DATA[94,3] := 2.0;
   DATA[94,4] := 261.9841;
   DATA[94,5] := 8.391951;
   DATA[94,6] := 328.4286;
   DATA[94,7] := 2.442188;
   DATA[94,8] := 2.0;
   DATA[94,9] := 2.0;
   DATA[94,10] := 2.0;
   DATA[94,11] := 19.65875;
   DATA[94,12] := 2.212343;
   DATA[94,13] := 960.0103;
   DATA[94,14] := 1.0;
   DATA[94,15] := 2.0;
   DATA[94,16] := 1.0;
   DATA[94,17] := 1.0;
   DATA[94,18] := 1.0;
   DATA[94,19] := 2.0;
   DATA[94,20] := 148.808;
   DATA[94,21] := 156.0882;
   DATA[94,22] := 1.714029;
   DATA[94,23] := 950.8331;
   DATA[94,24] := 2.0;
   DATA[94,25] := 2.0;
   DATA[94,26] := 7.877019;
   DATA[94,27] := 145.1423;
   DATA[94,28] := 264.2592;
   DATA[94,29] := 12.30454;
   DATA[94,30] := 1.727378;
   DATA[94,31] := 1.257589;
   DATA[94,32] := 0.7353967;
   DATA[94,33] := 0.3065048;
   DATA[94,34] := 2.0;
   DATA[94,35] := 251.1055;
   DATA[94,36] := 1.649953;
   DATA[94,37] := 189.7751;
   DATA[94,38] := 0.000128152;
   DATA[94,39] := 1.0;
   DATA[95,0] := 2.554847;
   DATA[95,1] := 527.3608;
   DATA[95,2] := 2.0;
   DATA[95,3] := 2.0;
   DATA[95,4] := 261.9841;
   DATA[95,5] := 8.391951;
   DATA[95,6] := 328.4286;
   DATA[95,7] := 2.442188;
   DATA[95,8] := 2.0;
   DATA[95,9] := 2.0;
   DATA[95,10] := 2.0;
   DATA[95,11] := 19.65875;
   DATA[95,12] := 2.212343;
   DATA[95,13] := 959.9302;
   DATA[95,14] := 1.0;
   DATA[95,15] := 2.0;
   DATA[95,16] := 1.0;
   DATA[95,17] := 1.0;
   DATA[95,18] := 1.0;
   DATA[95,19] := 2.0;
   DATA[95,20] := 148.808;
   DATA[95,21] := 156.0882;
   DATA[95,22] := 1.713261;
   DATA[95,23] := 950.91;
   DATA[95,24] := 2.0;
   DATA[95,25] := 2.0;
   DATA[95,26] := 7.877019;
   DATA[95,27] := 145.1423;
   DATA[95,28] := 264.2592;
   DATA[95,29] := 12.30454;
   DATA[95,30] := 1.727378;
   DATA[95,31] := 1.245549;
   DATA[95,32] := 0.7353967;
